   1:  PR[91,3] = PR[90,3] + 83.496;
   1:L PR[91] R[100]mm/sec CNT100;
   1:  PR[91,1] = PR[90,1] + -62.858;
   1:  PR[91,2] = PR[90,2] + -8.805;
   1:  PR[91,3] = PR[90,3] + 83.508;
   1:L PR[91] R[100]mm/sec CNT100;
   1:  PR[91,1] = PR[90,1] + -62.357;
   1:  PR[91,2] = PR[90,2] + -9.939;
   1:  PR[91,3] = PR[90,3] + 83.523;
   1:L PR[91] R[100]mm/sec CNT100;
   1:  PR[91,1] = PR[90,1] + -59.299;
   1:  PR[91,2] = PR[90,2] + -14.135;
   1:  PR[91,3] = PR[90,3] + 83.529;
   1:L PR[91] R[100]mm/sec CNT100;
   1:  PR[91,1] = PR[90,1] + -58.899;
   1:  PR[91,2] = PR[90,2] + -14.496;
   1:  PR[91,3] = PR[90,3] + 83.550;
   1:L PR[91] R[100]mm/sec CNT100;
   1:  PR[91,1] = PR[90,1] + -55.480;
   1:  PR[91,2] = PR[90,2] + -17.247;
   1:  PR[91,3] = PR[90,3] + 83.552;
   1:L PR[91] R[100]mm/sec CNT100;
   1:  PR[91,1] = PR[90,1] + -54.310;
   1:  PR[91,2] = PR[90,2] + -18.147;
   1:  PR[91,3] = PR[90,3] + 83.570;
   1:L PR[91] R[100]mm/sec CNT100;
   1:  PR[91,1] = PR[90,1] + -51.181;
   1:  PR[91,2] = PR[90,2] + -19.877;
   1:  PR[91,3] = PR[90,3] + 83.576;
   1:L PR[91] R[100]mm/sec CNT100;
   1:  PR[91,1] = PR[90,1] + -47.305;
   1:  PR[91,2] = PR[90,2] + -21.893;
   1:  PR[91,3] = PR[90,3] + 83.591;
   1:L PR[91] R[100]mm/sec CNT100;
   1:  PR[91,1] = PR[90,1] + -46.433;
   1:  PR[91,2] = PR[90,2] + -22.219;
   1:  PR[91,3] = PR[90,3] + 83.609;
   1:L PR[91] R[100]mm/sec CNT100;
   1:  PR[91,1] = PR[90,1] + -44.851;
   1:  PR[91,2] = PR[90,2] + -22.759;
   1:  PR[91,3] = PR[90,3] + 83.613;
   1:L PR[91] R[100]mm/sec CNT100;
   1:  PR[91,1] = PR[90,1] + -40.571;
   1:  PR[91,2] = PR[90,2] + -24.060;
   1:  PR[91,3] = PR[90,3] + 83.620;
   1:L PR[91] R[100]mm/sec CNT100;
   1:  PR[91,1] = PR[90,1] + -38.296;
   1:  PR[91,2] = PR[90,2] + -24.719;
   1:  PR[91,3] = PR[90,3] + 83.638;
   1:L PR[91] R[100]mm/sec CNT100;
   1:  PR[91,1] = PR[90,1] + -32.592;
   1:  PR[91,2] = PR[90,2] + -25.826;
   1:  PR[91,3] = PR[90,3] + 83.648;
   1:L PR[91] R[100]mm/sec CNT100;
   1:  PR[91,1] = PR[90,1] + -30.326;
   1:  PR[91,2] = PR[90,2] + -26.230;
   1:  PR[91,3] = PR[90,3] + 83.672;
   1:L PR[91] R[100]mm/sec CNT100;
   1:  PR[91,1] = PR[90,1] + -20.814;
   1:  PR[91,2] = PR[90,2] + -27.225;
   1:  PR[91,3] = PR[90,3] + 83.681;
   1:L PR[91] R[100]mm/sec CNT100;
   1:  PR[91,1] = PR[90,1] + -17.150;
   1:  PR[91,2] = PR[90,2] + -27.366;
   1:  PR[91,3] = PR[90,3] + 83.721;
   1:L PR[91] R[100]mm/sec CNT100;
   1:  PR[91,1] = PR[90,1] + -10.849;
   1:  PR[91,2] = PR[90,2] + -27.576;
   1:  PR[91,3] = PR[90,3] + 83.736;
   1:L PR[91] R[100]mm/sec CNT100;
   1:  PR[91,1] = PR[90,1] + -4.026;
   1:  PR[91,2] = PR[90,2] + -27.361;
   1:  PR[91,3] = PR[90,3] + 83.762;
   1:L PR[91] R[100]mm/sec CNT100;
   1:  PR[91,1] = PR[90,1] + -0.594;
   1:  PR[91,2] = PR[90,2] + -27.232;
   1:  PR[91,3] = PR[90,3] + 83.790;
   1:L PR[91] R[100]mm/sec CNT100;
   1:  PR[91,1] = PR[90,1] + 0.853;
   1:  PR[91,2] = PR[90,2] + -27.123;
   1:  PR[91,3] = PR[90,3] + 83.804;
   1:L PR[91] R[100]mm/sec CNT100;
   1:  PR[91,1] = PR[90,1] + 2.653;
   1:  PR[91,2] = PR[90,2] + -27.252;
   1:  PR[91,3] = PR[90,3] + 83.810;
   1:L PR[91] R[100]mm/sec CNT100;
   1:  PR[91,1] = PR[90,1] + 5.506;
   1:  PR[91,2] = PR[90,2] + -27.258;
   1:  PR[91,3] = PR[90,3] + 83.818;
   1:L PR[91] R[100]mm/sec CNT100;
   1:  PR[91,1] = PR[90,1] + 7.419;
   1:  PR[91,2] = PR[90,2] + -27.285;
   1:  PR[91,3] = PR[90,3] + 83.829;
   1:L PR[91] R[100]mm/sec CNT100;
   1:  PR[91,1] = PR[90,1] + 7.750;
   1:  PR[91,2] = PR[90,2] + -27.279;
   1:  PR[91,3] = PR[90,3] + 83.837;
   1:L PR[91] R[100]mm/sec CNT100;
   1:  PR[91,1] = PR[90,1] + 8.440;
   1:  PR[91,2] = PR[90,2] + -27.232;
   1:  PR[91,3] = PR[90,3] + 83.839;
   1:L PR[91] R[100]mm/sec CNT100;
   1:  PR[91,1] = PR[90,1] + 11.886;
   1:  PR[91,2] = PR[90,2] + -26.903;
   1:  PR[91,3] = PR[90,3] + 83.841;
   1:L PR[91] R[100]mm/sec CNT100;
   1:  PR[91,1] = PR[90,1] + 12.853;
   1:  PR[91,2] = PR[90,2] + -27.102;
   1:  PR[91,3] = PR[90,3] + 83.856;
   1:L PR[91] R[100]mm/sec CNT100;
   1:  PR[91,1] = PR[90,1] + 15.186;
   1:  PR[91,2] = PR[90,2] + -27.492;
   1:  PR[91,3] = PR[90,3] + 83.860;
   1:L PR[91] R[100]mm/sec CNT100;
   1:  PR[91,1] = PR[90,1] + 17.292;
   1:  PR[91,2] = PR[90,2] + -27.750;
   1:  PR[91,3] = PR[90,3] + 83.870;
   1:L PR[91] R[100]mm/sec CNT100;
   1:  PR[91,1] = PR[90,1] + 20.645;
   1:  PR[91,2] = PR[90,2] + -27.636;
   1:  PR[91,3] = PR[90,3] + 83.878;
   1:L PR[91] R[100]mm/sec CNT100;
   1:  PR[91,1] = PR[90,1] + 22.928;
   1:  PR[91,2] = PR[90,2] + -27.593;
   1:  PR[91,3] = PR[90,3] + 83.892;
   1:L PR[91] R[100]mm/sec CNT100;
   1:  PR[91,1] = PR[90,1] + 26.835;
   1:  PR[91,2] = PR[90,2] + -28.529;
   1:  PR[91,3] = PR[90,3] + 83.901;
   1:L PR[91] R[100]mm/sec CNT100;
   1:  PR[91,1] = PR[90,1] + 28.431;
   1:  PR[91,2] = PR[90,2] + -28.891;
   1:  PR[91,3] = PR[90,3] + 83.918;
   1:L PR[91] R[100]mm/sec CNT100;
   1:  PR[91,1] = PR[90,1] + 33.590;
   1:  PR[91,2] = PR[90,2] + -29.193;
   1:  PR[91,3] = PR[90,3] + 83.925;
   1:L PR[91] R[100]mm/sec CNT100;
   1:  PR[91,1] = PR[90,1] + 38.798;
   1:  PR[91,2] = PR[90,2] + -28.611;
   1:  PR[91,3] = PR[90,3] + 83.946;
   1:L PR[91] R[100]mm/sec CNT100;
   1:  PR[91,1] = PR[90,1] + 41.367;
   1:  PR[91,2] = PR[90,2] + -27.900;
   1:  PR[91,3] = PR[90,3] + 83.968;
   1:L PR[91] R[100]mm/sec CNT100;
   1:  PR[91,1] = PR[90,1] + 43.735;
   1:  PR[91,2] = PR[90,2] + -27.217;
   1:  PR[91,3] = PR[90,3] + 83.979;
   1:L PR[91] R[100]mm/sec CNT100;
   1:  PR[91,1] = PR[90,1] + 47.721;
   1:  PR[91,2] = PR[90,2] + -25.319;
   1:  PR[91,3] = PR[90,3] + 83.989;
   1:L PR[91] R[100]mm/sec CNT100;
   1:  PR[91,1] = PR[90,1] + 48.381;
   1:  PR[91,2] = PR[90,2] + -25.044;
   1:  PR[91,3] = PR[90,3] + 84.007;
   1:L PR[91] R[100]mm/sec CNT100;
   1:  PR[91,1] = PR[90,1] + 48.578;
   1:  PR[91,2] = PR[90,2] + -24.941;
   1:  PR[91,3] = PR[90,3] + 84.010;
   1:L PR[91] R[100]mm/sec CNT100;
   1:  PR[91,1] = PR[90,1] + 51.923;
   1:  PR[91,2] = PR[90,2] + -22.835;
   1:  PR[91,3] = PR[90,3] + 84.011;
   1:L PR[91] R[100]mm/sec CNT100;
   1:  PR[91,1] = PR[90,1] + 53.939;
   1:  PR[91,2] = PR[90,2] + -21.330;
   1:  PR[91,3] = PR[90,3] + 84.027;
   1:L PR[91] R[100]mm/sec CNT100;
   1:  PR[91,1] = PR[90,1] + 54.792;
   1:  PR[91,2] = PR[90,2] + -20.561;
   1:  PR[91,3] = PR[90,3] + 84.037;
   1:L PR[91] R[100]mm/sec CNT100;
   1:  PR[91,1] = PR[90,1] + 56.133;
   1:  PR[91,2] = PR[90,2] + -19.163;
   1:  PR[91,3] = PR[90,3] + 84.042;
   1:L PR[91] R[100]mm/sec CNT100;
   1:  PR[91,1] = PR[90,1] + 57.720;
   1:  PR[91,2] = PR[90,2] + -17.820;
   1:  PR[91,3] = PR[90,3] + 84.050;
   1:L PR[91] R[100]mm/sec CNT100;
   1:  PR[91,1] = PR[90,1] + 58.592;
   1:  PR[91,2] = PR[90,2] + -16.934;
   1:  PR[91,3] = PR[90,3] + 84.059;
   1:L PR[91] R[100]mm/sec CNT100;
   1:  PR[91,1] = PR[90,1] + 60.063;
   1:  PR[91,2] = PR[90,2] + -15.177;
   1:  PR[91,3] = PR[90,3] + 84.064;
   1:L PR[91] R[100]mm/sec CNT100;
   1:  PR[91,1] = PR[90,1] + 61.896;
   1:  PR[91,2] = PR[90,2] + -12.606;
   1:  PR[91,3] = PR[90,3] + 84.073;
   1:L PR[91] R[100]mm/sec CNT100;
   1:  PR[91,1] = PR[90,1] + 62.073;
   1:  PR[91,2] = PR[90,2] + -12.393;
   1:  PR[91,3] = PR[90,3] + 84.086;
   1:L PR[91] R[100]mm/sec CNT100;
   1:  PR[91,1] = PR[90,1] + 62.111;
   1:  PR[91,2] = PR[90,2] + -12.327;
   1:  PR[91,3] = PR[90,3] + 84.087;
   1:L PR[91] R[100]mm/sec CNT100;
   1:  PR[91,1] = PR[90,1] + 64.147;
   1:  PR[91,2] = PR[90,2] + -8.707;
   1:  PR[91,3] = PR[90,3] + 84.088;
   1:L PR[91] R[100]mm/sec CNT100;
   1:  PR[91,1] = PR[90,1] + 64.790;
   1:  PR[91,2] = PR[90,2] + -6.800;
   1:  PR[91,3] = PR[90,3] + 84.105;
   1:L PR[91] R[100]mm/sec CNT100;
   1:  PR[91,1] = PR[90,1] + 65.448;
   1:  PR[91,2] = PR[90,2] + -4.780;
   1:  PR[91,3] = PR[90,3] + 84.113;
   1:L PR[91] R[100]mm/sec CNT100;
   1:  PR[91,1] = PR[90,1] + 65.893;
   1:  PR[91,2] = PR[90,2] + -0.729;
   1:  PR[91,3] = PR[90,3] + 84.122;
   1:L PR[91] R[100]mm/sec CNT100;
   1:  PR[91,1] = PR[90,1] + 65.448;
   1:  PR[91,2] = PR[90,2] + 3.322;
   1:  PR[91,3] = PR[90,3] + 84.139;
   1:L PR[91] R[100]mm/sec CNT100;
   1:  PR[91,1] = PR[90,1] + 64.790;
   1:  PR[91,2] = PR[90,2] + 5.341;
   1:  PR[91,3] = PR[90,3] + 84.156;
   1:L PR[91] R[100]mm/sec CNT100;
   1:  PR[91,1] = PR[90,1] + 64.147;
   1:  PR[91,2] = PR[90,2] + 7.247;
   1:  PR[91,3] = PR[90,3] + 84.164;
   1:L PR[91] R[100]mm/sec CNT100;
   1:  PR[91,1] = PR[90,1] + 62.065;
   1:  PR[91,2] = PR[90,2] + 10.944;
   1:  PR[91,3] = PR[90,3] + 84.173;
   1:L PR[91] R[100]mm/sec CNT100;
   1:  PR[91,1] = PR[90,1] + 61.896;
   1:  PR[91,2] = PR[90,2] + 11.147;
   1:  PR[91,3] = PR[90,3] + 84.190;
   1:L PR[91] R[100]mm/sec CNT100;
   1:  PR[91,1] = PR[90,1] + 60.063;
   1:  PR[91,2] = PR[90,2] + 13.718;
   1:  PR[91,3] = PR[90,3] + 84.191;
   1:L PR[91] R[100]mm/sec CNT100;
   1:  PR[91,1] = PR[90,1] + 58.592;
   1:  PR[91,2] = PR[90,2] + 15.476;
   1:  PR[91,3] = PR[90,3] + 84.204;
   1:L PR[91] R[100]mm/sec CNT100;
   1:  PR[91,1] = PR[90,1] + 57.720;
   1:  PR[91,2] = PR[90,2] + 16.362;
   1:  PR[91,3] = PR[90,3] + 84.214;
   1:L PR[91] R[100]mm/sec CNT100;
   1:  PR[91,1] = PR[90,1] + 56.133;
   1:  PR[91,2] = PR[90,2] + 17.704;
   1:  PR[91,3] = PR[90,3] + 84.219;
   1:L PR[91] R[100]mm/sec CNT100;
   1:  PR[91,1] = PR[90,1] + 54.792;
   1:  PR[91,2] = PR[90,2] + 19.102;
   1:  PR[91,3] = PR[90,3] + 84.227;
   1:L PR[91] R[100]mm/sec CNT100;
   1:  PR[91,1] = PR[90,1] + 53.939;
   1:  PR[91,2] = PR[90,2] + 19.872;
   1:  PR[91,3] = PR[90,3] + 84.235;
   1:L PR[91] R[100]mm/sec CNT100;
   1:  PR[91,1] = PR[90,1] + 51.923;
   1:  PR[91,2] = PR[90,2] + 21.376;
   1:  PR[91,3] = PR[90,3] + 84.240;
   1:L PR[91] R[100]mm/sec CNT100;
   1:  PR[91,1] = PR[90,1] + 48.578;
   1:  PR[91,2] = PR[90,2] + 23.482;
   1:  PR[91,3] = PR[90,3] + 84.250;
   1:L PR[91] R[100]mm/sec CNT100;
   1:  PR[91,1] = PR[90,1] + 48.381;
   1:  PR[91,2] = PR[90,2] + 23.585;
   1:  PR[91,3] = PR[90,3] + 84.267;
   1:L PR[91] R[100]mm/sec CNT100;
   1:  PR[91,1] = PR[90,1] + 47.721;
   1:  PR[91,2] = PR[90,2] + 23.860;
   1:  PR[91,3] = PR[90,3] + 84.268;
   1:L PR[91] R[100]mm/sec CNT100;
   1:  PR[91,1] = PR[90,1] + 43.735;
   1:  PR[91,2] = PR[90,2] + 25.759;
   1:  PR[91,3] = PR[90,3] + 84.270;
   1:L PR[91] R[100]mm/sec CNT100;
   1:  PR[91,1] = PR[90,1] + 41.367;
   1:  PR[91,2] = PR[90,2] + 26.441;
   1:  PR[91,3] = PR[90,3] + 84.289;
   1:L PR[91] R[100]mm/sec CNT100;
   1:  PR[91,1] = PR[90,1] + 38.798;
   1:  PR[91,2] = PR[90,2] + 27.152;
   1:  PR[91,3] = PR[90,3] + 84.299;
   1:L PR[91] R[100]mm/sec CNT100;
   1:  PR[91,1] = PR[90,1] + 33.590;
   1:  PR[91,2] = PR[90,2] + 27.734;
   1:  PR[91,3] = PR[90,3] + 84.310;
   1:L PR[91] R[100]mm/sec CNT100;
   1:  PR[91,1] = PR[90,1] + 28.431;
   1:  PR[91,2] = PR[90,2] + 27.432;
   1:  PR[91,3] = PR[90,3] + 84.331;
   1:L PR[91] R[100]mm/sec CNT100;
   1:  PR[91,1] = PR[90,1] + 26.835;
   1:  PR[91,2] = PR[90,2] + 27.070;
   1:  PR[91,3] = PR[90,3] + 84.353;
   1:L PR[91] R[100]mm/sec CNT100;
   1:  PR[91,1] = PR[90,1] + 22.911;
   1:  PR[91,2] = PR[90,2] + 26.131;
   1:  PR[91,3] = PR[90,3] + 84.359;
   1:L PR[91] R[100]mm/sec CNT100;
   1:  PR[91,1] = PR[90,1] + 19.492;
   1:  PR[91,2] = PR[90,2] + 26.252;
   1:  PR[91,3] = PR[90,3] + 84.376;
   1:L PR[91] R[100]mm/sec CNT100;
   1:  PR[91,1] = PR[90,1] + 17.308;
   1:  PR[91,2] = PR[90,2] + 26.293;
   1:  PR[91,3] = PR[90,3] + 84.390;
   1:L PR[91] R[100]mm/sec CNT100;
   1:  PR[91,1] = PR[90,1] + 15.188;
   1:  PR[91,2] = PR[90,2] + 26.034;
   1:  PR[91,3] = PR[90,3] + 84.399;
   1:L PR[91] R[100]mm/sec CNT100;
   1:  PR[91,1] = PR[90,1] + 12.855;
   1:  PR[91,2] = PR[90,2] + 25.644;
   1:  PR[91,3] = PR[90,3] + 84.408;
   1:L PR[91] R[100]mm/sec CNT100;
   1:  PR[91,1] = PR[90,1] + 11.886;
   1:  PR[91,2] = PR[90,2] + 25.445;
   1:  PR[91,3] = PR[90,3] + 84.418;
   1:L PR[91] R[100]mm/sec CNT100;
   1:  PR[91,1] = PR[90,1] + 8.440;
   1:  PR[91,2] = PR[90,2] + 25.773;
   1:  PR[91,3] = PR[90,3] + 84.422;
   1:L PR[91] R[100]mm/sec CNT100;
   1:  PR[91,1] = PR[90,1] + 7.775;
   1:  PR[91,2] = PR[90,2] + 25.818;
   1:  PR[91,3] = PR[90,3] + 84.436;
   1:L PR[91] R[100]mm/sec CNT100;
   1:  PR[91,1] = PR[90,1] + 2.699;
   1:  PR[91,2] = PR[90,2] + 25.794;
   1:  PR[91,3] = PR[90,3] + 84.439;
   1:L PR[91] R[100]mm/sec CNT100;
   1:  PR[91,1] = PR[90,1] + 1.042;
   1:  PR[91,2] = PR[90,2] + 25.626;
   1:  PR[91,3] = PR[90,3] + 84.460;
   1:L PR[91] R[100]mm/sec CNT100;
   1:  PR[91,1] = PR[90,1] + 0.458;
   1:  PR[91,2] = PR[90,2] + 25.698;
   1:  PR[91,3] = PR[90,3] + 84.467;
   1:L PR[91] R[100]mm/sec CNT100;
   1:  PR[91,1] = PR[90,1] + -0.211;
   1:  PR[91,2] = PR[90,2] + 25.747;
   1:  PR[91,3] = PR[90,3] + 84.469;
   1:L PR[91] R[100]mm/sec CNT100;
   1:  PR[91,1] = PR[90,1] + -4.029;
   1:  PR[91,2] = PR[90,2] + 25.902;
   1:  PR[91,3] = PR[90,3] + 84.472;
   1:L PR[91] R[100]mm/sec CNT100;
   1:  PR[91,1] = PR[90,1] + -10.849;
   1:  PR[91,2] = PR[90,2] + 26.117;
   1:  PR[91,3] = PR[90,3] + 84.487;
   1:L PR[91] R[100]mm/sec CNT100;
   1:  PR[91,1] = PR[90,1] + -17.150;
   1:  PR[91,2] = PR[90,2] + 25.907;
   1:  PR[91,3] = PR[90,3] + 84.516;
   1:L PR[91] R[100]mm/sec CNT100;
   1:  PR[91,1] = PR[90,1] + -20.814;
   1:  PR[91,2] = PR[90,2] + 25.766;
   1:  PR[91,3] = PR[90,3] + 84.542;
   1:L PR[91] R[100]mm/sec CNT100;
   1:  PR[91,1] = PR[90,1] + -30.326;
   1:  PR[91,2] = PR[90,2] + 24.771;
   1:  PR[91,3] = PR[90,3] + 84.557;
   1:L PR[91] R[100]mm/sec CNT100;
   1:  PR[91,1] = PR[90,1] + -32.592;
   1:  PR[91,2] = PR[90,2] + 24.367;
   1:  PR[91,3] = PR[90,3] + 84.596;
   1:L PR[91] R[100]mm/sec CNT100;
   1:  PR[91,1] = PR[90,1] + -38.503;
   1:  PR[91,2] = PR[90,2] + 23.224;
   1:  PR[91,3] = PR[90,3] + 84.606;
   1:L PR[91] R[100]mm/sec CNT100;
   1:  PR[91,1] = PR[90,1] + -43.527;
   1:  PR[91,2] = PR[90,2] + 21.723;
   1:  PR[91,3] = PR[90,3] + 84.630;
   1:L PR[91] R[100]mm/sec CNT100;
   1:  PR[91,1] = PR[90,1] + -46.770;
   1:  PR[91,2] = PR[90,2] + 20.639;
   1:  PR[91,3] = PR[90,3] + 84.652;
   1:L PR[91] R[100]mm/sec CNT100;
   1:  PR[91,1] = PR[90,1] + -50.439;
   1:  PR[91,2] = PR[90,2] + 18.870;
   1:  PR[91,3] = PR[90,3] + 84.666;
   1:L PR[91] R[100]mm/sec CNT100;
   1:  PR[91,1] = PR[90,1] + -53.072;
   1:  PR[91,2] = PR[90,2] + 17.528;
   1:  PR[91,3] = PR[90,3] + 84.683;
   1:L PR[91] R[100]mm/sec CNT100;
   1:  PR[91] = PR[90];
   1:  PR[91,1] = PR[90,1] + -56.871;
   1:  PR[91,2] = PR[90,2] + 13.843;
   1:  PR[91,3] = PR[90,3] + 85.995;
   1:L PR[91] R[100]mm/sec CNT100;
   1:  PR[91,1] = PR[90,1] + -57.057;
   1:  PR[91,2] = PR[90,2] + 13.694;
   1:  PR[91,3] = PR[90,3] + 84.721;
   1:L PR[91] R[100]mm/sec CNT100;
   1:  PR[91,1] = PR[90,1] + -60.068;
   1:  PR[91,2] = PR[90,2] + 10.000;
   1:  PR[91,3] = PR[90,3] + 84.722;
   1:L PR[91] R[100]mm/sec CNT100;
   1:  PR[91,1] = PR[90,1] + -60.841;
   1:  PR[91,2] = PR[90,2] + 9.015;
   1:  PR[91,3] = PR[90,3] + 84.742;
   1:L PR[91] R[100]mm/sec CNT100;
   1:  PR[91,1] = PR[90,1] + -62.232;
   1:  PR[91,2] = PR[90,2] + 5.989;
   1:  PR[91,3] = PR[90,3] + 84.747;
   1:L PR[91] R[100]mm/sec CNT100;
   1:  PR[91,1] = PR[90,1] + -63.043;
   1:  PR[91,2] = PR[90,2] + 4.170;
   1:  PR[91,3] = PR[90,3] + 84.761;
   1:L PR[91] R[100]mm/sec CNT100;
   1:  PR[91,1] = PR[90,1] + -63.397;
   1:  PR[91,2] = PR[90,2] + 1.755;
   1:  PR[91,3] = PR[90,3] + 84.770;
   1:L PR[91] R[100]mm/sec CNT100;
   1:  PR[91,1] = PR[90,1] + -63.845;
   1:  PR[91,2] = PR[90,2] + -0.138;
   1:  PR[91,3] = PR[90,3] + 84.780;
   1:L PR[91] R[100]mm/sec CNT100;
   1:  PR[91,1] = PR[90,1] + -63.928;
   1:  PR[91,2] = PR[90,2] + -0.626;
   1:  PR[91,3] = PR[90,3] + 84.788;
   1:L PR[91] R[100]mm/sec CNT100;
   1:  PR[91,1] = PR[90,1] + -63.631;
   1:  PR[91,2] = PR[90,2] + -1.695;
   1:  PR[91,3] = PR[90,3] + 84.790;
   1:L PR[91] R[100]mm/sec CNT100;
   1:  PR[91,1] = PR[90,1] + -63.134;
   1:  PR[91,2] = PR[90,2] + -5.424;
   1:  PR[91,3] = PR[90,3] + 84.795;
   1:L PR[91] R[100]mm/sec CNT100;
   1:  PR[91,1] = PR[90,1] + -61.433;
   1:  PR[91,2] = PR[90,2] + -9.549;
   1:  PR[91,3] = PR[90,3] + 84.810;
   1:L PR[91] R[100]mm/sec CNT100;
   1:  PR[91,1] = PR[90,1] + -61.268;
   1:  PR[91,2] = PR[90,2] + -9.923;
   1:  PR[91,3] = PR[90,3] + 84.829;
   1:L PR[91] R[100]mm/sec CNT100;
   1:  PR[91,1] = PR[90,1] + -59.724;
   1:  PR[91,2] = PR[90,2] + -12.049;
   1:  PR[91,3] = PR[90,3] + 84.831;
   1:L PR[91] R[100]mm/sec CNT100;
   1:  PR[91,1] = PR[90,1] + -57.969;
   1:  PR[91,2] = PR[90,2] + -14.174;
   1:  PR[91,3] = PR[90,3] + 84.842;
   1:L PR[91] R[100]mm/sec CNT100;
   1:  PR[91,1] = PR[90,1] + -54.587;
   1:  PR[91,2] = PR[90,2] + -16.895;
   1:  PR[91,3] = PR[90,3] + 84.853;
   1:L PR[91] R[100]mm/sec CNT100;
   1:  PR[91,1] = PR[90,1] + -52.665;
   1:  PR[91,2] = PR[90,2] + -18.373;
   1:  PR[91,3] = PR[90,3] + 84.871;
   1:L PR[91] R[100]mm/sec CNT100;
   1:  PR[91,1] = PR[90,1] + -50.363;
   1:  PR[91,2] = PR[90,2] + -19.646;
   1:  PR[91,3] = PR[90,3] + 84.881;
   1:L PR[91] R[100]mm/sec CNT100;
   1:  PR[91,1] = PR[90,1] + -45.579;
   1:  PR[91,2] = PR[90,2] + -22.133;
   1:  PR[91,3] = PR[90,3] + 84.892;
   1:L PR[91] R[100]mm/sec CNT100;
   1:  PR[91,1] = PR[90,1] + -39.579;
   1:  PR[91,2] = PR[90,2] + -23.958;
   1:  PR[91,3] = PR[90,3] + 84.915;
   1:L PR[91] R[100]mm/sec CNT100;
   1:  PR[91,1] = PR[90,1] + -36.288;
   1:  PR[91,2] = PR[90,2] + -24.911;
   1:  PR[91,3] = PR[90,3] + 84.941;
   1:L PR[91] R[100]mm/sec CNT100;
   1:  PR[91,1] = PR[90,1] + -33.240;
   1:  PR[91,2] = PR[90,2] + -25.503;
   1:  PR[91,3] = PR[90,3] + 84.955;
   1:L PR[91] R[100]mm/sec CNT100;
   1:  PR[91,1] = PR[90,1] + -27.855;
   1:  PR[91,2] = PR[90,2] + -26.462;
   1:  PR[91,3] = PR[90,3] + 84.968;
   1:L PR[91] R[100]mm/sec CNT100;
   1:  PR[91,1] = PR[90,1] + -18.268;
   1:  PR[91,2] = PR[90,2] + -27.470;
   1:  PR[91,3] = PR[90,3] + 84.991;
   1:L PR[91] R[100]mm/sec CNT100;
   1:  PR[91,1] = PR[90,1] + -13.610;
   1:  PR[91,2] = PR[90,2] + -27.649;
   1:  PR[91,3] = PR[90,3] + 85.031;
   1:L PR[91] R[100]mm/sec CNT100;
   1:  PR[91,1] = PR[90,1] + -8.222;
   1:  PR[91,2] = PR[90,2] + -27.828;
   1:  PR[91,3] = PR[90,3] + 85.051;
   1:L PR[91] R[100]mm/sec CNT100;
   1:  PR[91,1] = PR[90,1] + -0.378;
   1:  PR[91,2] = PR[90,2] + -27.581;
   1:  PR[91,3] = PR[90,3] + 85.073;
   1:L PR[91] R[100]mm/sec CNT100;
   1:  PR[91,1] = PR[90,1] + 2.123;
   1:  PR[91,2] = PR[90,2] + -27.487;
   1:  PR[91,3] = PR[90,3] + 85.106;
   1:L PR[91] R[100]mm/sec CNT100;
   1:  PR[91,1] = PR[90,1] + 2.862;
   1:  PR[91,2] = PR[90,2] + -27.436;
   1:  PR[91,3] = PR[90,3] + 85.116;
   1:L PR[91] R[100]mm/sec CNT100;
   1:  PR[91,1] = PR[90,1] + 3.357;
   1:  PR[91,2] = PR[90,2] + -27.468;
   1:  PR[91,3] = PR[90,3] + 85.119;
   1:L PR[91] R[100]mm/sec CNT100;
   1:  PR[91,1] = PR[90,1] + 7.999;
   1:  PR[91,2] = PR[90,2] + -27.526;
   1:  PR[91,3] = PR[90,3] + 85.122;
   1:L PR[91] R[100]mm/sec CNT100;
   1:  PR[91,1] = PR[90,1] + 8.784;
   1:  PR[91,2] = PR[90,2] + -27.509;
   1:  PR[91,3] = PR[90,3] + 85.141;
   1:L PR[91] R[100]mm/sec CNT100;
   1:  PR[91,1] = PR[90,1] + 10.312;
   1:  PR[91,2] = PR[90,2] + -27.406;
   1:  PR[91,3] = PR[90,3] + 85.144;
   1:L PR[91] R[100]mm/sec CNT100;
   1:  PR[91,1] = PR[90,1] + 12.488;
   1:  PR[91,2] = PR[90,2] + -27.206;
   1:  PR[91,3] = PR[90,3] + 85.151;
   1:L PR[91] R[100]mm/sec CNT100;
   1:  PR[91,1] = PR[90,1] + 14.691;
   1:  PR[91,2] = PR[90,2] + -27.574;
   1:  PR[91,3] = PR[90,3] + 85.160;
   1:L PR[91] R[100]mm/sec CNT100;
   1:  PR[91,1] = PR[90,1] + 17.503;
   1:  PR[91,2] = PR[90,2] + -27.919;
   1:  PR[91,3] = PR[90,3] + 85.169;
   1:L PR[91] R[100]mm/sec CNT100;
   1:  PR[91,1] = PR[90,1] + 19.520;
   1:  PR[91,2] = PR[90,2] + -27.850;
   1:  PR[91,3] = PR[90,3] + 85.181;
   1:L PR[91] R[100]mm/sec CNT100;
   1:  PR[91,1] = PR[90,1] + 22.617;
   1:  PR[91,2] = PR[90,2] + -27.793;
   1:  PR[91,3] = PR[90,3] + 85.189;
   1:L PR[91] R[100]mm/sec CNT100;
   1:  PR[91,1] = PR[90,1] + 25.077;
   1:  PR[91,2] = PR[90,2] + -28.382;
   1:  PR[91,3] = PR[90,3] + 85.202;
   1:L PR[91] R[100]mm/sec CNT100;
   1:  PR[91,1] = PR[90,1] + 26.255;
   1:  PR[91,2] = PR[90,2] + -28.638;
   1:  PR[91,3] = PR[90,3] + 85.213;
   1:L PR[91] R[100]mm/sec CNT100;
   1:  PR[91,1] = PR[90,1] + 28.183;
   1:  PR[91,2] = PR[90,2] + -29.086;
   1:  PR[91,3] = PR[90,3] + 85.218;
   1:L PR[91] R[100]mm/sec CNT100;
   1:  PR[91,1] = PR[90,1] + 33.328;
   1:  PR[91,2] = PR[90,2] + -29.386;
   1:  PR[91,3] = PR[90,3] + 85.226;
   1:L PR[91] R[100]mm/sec CNT100;
   1:  PR[91,1] = PR[90,1] + 35.825;
   1:  PR[91,2] = PR[90,2] + -29.084;
   1:  PR[91,3] = PR[90,3] + 85.247;
   1:L PR[91] R[100]mm/sec CNT100;
   1:  PR[91,1] = PR[90,1] + 38.494;
   1:  PR[91,2] = PR[90,2] + -28.783;
   1:  PR[91,3] = PR[90,3] + 85.258;
   1:L PR[91] R[100]mm/sec CNT100;
   1:  PR[91,1] = PR[90,1] + 39.496;
   1:  PR[91,2] = PR[90,2] + -28.506;
   1:  PR[91,3] = PR[90,3] + 85.269;
   1:L PR[91] R[100]mm/sec CNT100;
   1:  PR[91,1] = PR[90,1] + 43.463;
   1:  PR[91,2] = PR[90,2] + -27.362;
   1:  PR[91,3] = PR[90,3] + 85.273;
   1:L PR[91] R[100]mm/sec CNT100;
   1:  PR[91,1] = PR[90,1] + 48.032;
   1:  PR[91,2] = PR[90,2] + -25.178;
   1:  PR[91,3] = PR[90,3] + 85.291;
   1:L PR[91] R[100]mm/sec CNT100;
   1:  PR[91,1] = PR[90,1] + 49.734;
   1:  PR[91,2] = PR[90,2] + -23.962;
   1:  PR[91,3] = PR[90,3] + 85.312;
   1:L PR[91] R[100]mm/sec CNT100;
   1:  PR[91,1] = PR[90,1] + 51.975;
   1:  PR[91,2] = PR[90,2] + -22.551;
   1:  PR[91,3] = PR[90,3] + 85.321;
   1:L PR[91] R[100]mm/sec CNT100;
   1:  PR[91,1] = PR[90,1] + 52.913;
   1:  PR[91,2] = PR[90,2] + -21.851;
   1:  PR[91,3] = PR[90,3] + 85.332;
   1:L PR[91] R[100]mm/sec CNT100;
   1:  PR[91,1] = PR[90,1] + 54.901;
   1:  PR[91,2] = PR[90,2] + -20.057;
   1:  PR[91,3] = PR[90,3] + 85.336;
   1:L PR[91] R[100]mm/sec CNT100;
   1:  PR[91,1] = PR[90,1] + 57.147;
   1:  PR[91,2] = PR[90,2] + -17.716;
   1:  PR[91,3] = PR[90,3] + 85.348;
   1:L PR[91] R[100]mm/sec CNT100;
   1:  PR[91,1] = PR[90,1] + 57.233;
   1:  PR[91,2] = PR[90,2] + -17.604;
   1:  PR[91,3] = PR[90,3] + 85.361;
   1:L PR[91] R[100]mm/sec CNT100;
   1:  PR[91,1] = PR[90,1] + 57.549;
   1:  PR[91,2] = PR[90,2] + -17.139;
   1:  PR[91,3] = PR[90,3] + 85.362;
   1:L PR[91] R[100]mm/sec CNT100;
   1:  PR[91,1] = PR[90,1] + 59.784;
   1:  PR[91,2] = PR[90,2] + -14.469;
   1:  PR[91,3] = PR[90,3] + 85.364;
   1:L PR[91] R[100]mm/sec CNT100;
   1:  PR[91,1] = PR[90,1] + 60.799;
   1:  PR[91,2] = PR[90,2] + -13.045;
   1:  PR[91,3] = PR[90,3] + 85.379;
   1:L PR[91] R[100]mm/sec CNT100;
   1:  PR[91,1] = PR[90,1] + 61.561;
   1:  PR[91,2] = PR[90,2] + -11.686;
   1:  PR[91,3] = PR[90,3] + 85.386;
   1:L PR[91] R[100]mm/sec CNT100;
   1:  PR[91,1] = PR[90,1] + 62.905;
   1:  PR[91,2] = PR[90,2] + -8.916;
   1:  PR[91,3] = PR[90,3] + 85.392;
   1:L PR[91] R[100]mm/sec CNT100;
   1:  PR[91,1] = PR[90,1] + 63.054;
   1:  PR[91,2] = PR[90,2] + -8.651;
   1:  PR[91,3] = PR[90,3] + 85.405;
   1:L PR[91] R[100]mm/sec CNT100;
   1:  PR[91,1] = PR[90,1] + 64.327;
   1:  PR[91,2] = PR[90,2] + -4.746;
   1:  PR[91,3] = PR[90,3] + 85.407;
   1:L PR[91] R[100]mm/sec CNT100;
   1:  PR[91,1] = PR[90,1] + 64.762;
   1:  PR[91,2] = PR[90,2] + -0.729;
   1:  PR[91,3] = PR[90,3] + 85.424;
   1:L PR[91] R[100]mm/sec CNT100;
   1:  PR[91,1] = PR[90,1] + 64.327;
   1:  PR[91,2] = PR[90,2] + 3.287;
   1:  PR[91,3] = PR[90,3] + 85.441;
   1:L PR[91] R[100]mm/sec CNT100;
   1:  PR[91,1] = PR[90,1] + 63.054;
   1:  PR[91,2] = PR[90,2] + 7.192;
   1:  PR[91,3] = PR[90,3] + 85.457;
   1:L PR[91] R[100]mm/sec CNT100;
   1:  PR[91,1] = PR[90,1] + 62.905;
   1:  PR[91,2] = PR[90,2] + 7.457;
   1:  PR[91,3] = PR[90,3] + 85.474;
   1:L PR[91] R[100]mm/sec CNT100;
   1:  PR[91,1] = PR[90,1] + 61.561;
   1:  PR[91,2] = PR[90,2] + 10.227;
   1:  PR[91,3] = PR[90,3] + 85.476;
   1:L PR[91] R[100]mm/sec CNT100;
   1:  PR[91,1] = PR[90,1] + 60.799;
   1:  PR[91,2] = PR[90,2] + 11.587;
   1:  PR[91,3] = PR[90,3] + 85.489;
   1:L PR[91] R[100]mm/sec CNT100;
   1:  PR[91,1] = PR[90,1] + 59.784;
   1:  PR[91,2] = PR[90,2] + 13.010;
   1:  PR[91,3] = PR[90,3] + 85.495;
   1:L PR[91] R[100]mm/sec CNT100;
   1:  PR[91,1] = PR[90,1] + 57.549;
   1:  PR[91,2] = PR[90,2] + 15.680;
   1:  PR[91,3] = PR[90,3] + 85.502;
   1:L PR[91] R[100]mm/sec CNT100;
   1:  PR[91,1] = PR[90,1] + 57.233;
   1:  PR[91,2] = PR[90,2] + 16.145;
   1:  PR[91,3] = PR[90,3] + 85.517;
   1:L PR[91] R[100]mm/sec CNT100;
   1:  PR[91,1] = PR[90,1] + 57.147;
   1:  PR[91,2] = PR[90,2] + 16.257;
   1:  PR[91,3] = PR[90,3] + 85.519;
   1:L PR[91] R[100]mm/sec CNT100;
   1:  PR[91,1] = PR[90,1] + 54.901;
   1:  PR[91,2] = PR[90,2] + 18.599;
   1:  PR[91,3] = PR[90,3] + 85.520;
   1:L PR[91] R[100]mm/sec CNT100;
   1:  PR[91,1] = PR[90,1] + 52.913;
   1:  PR[91,2] = PR[90,2] + 20.392;
   1:  PR[91,3] = PR[90,3] + 85.533;
   1:L PR[91] R[100]mm/sec CNT100;
   1:  PR[91,1] = PR[90,1] + 51.975;
   1:  PR[91,2] = PR[90,2] + 21.092;
   1:  PR[91,3] = PR[90,3] + 85.545;
   1:L PR[91] R[100]mm/sec CNT100;
   1:  PR[91,1] = PR[90,1] + 49.734;
   1:  PR[91,2] = PR[90,2] + 22.503;
   1:  PR[91,3] = PR[90,3] + 85.549;
   1:L PR[91] R[100]mm/sec CNT100;
   1:  PR[91,1] = PR[90,1] + 48.032;
   1:  PR[91,2] = PR[90,2] + 23.719;
   1:  PR[91,3] = PR[90,3] + 85.560;
   1:L PR[91] R[100]mm/sec CNT100;
   1:  PR[91,1] = PR[90,1] + 43.463;
   1:  PR[91,2] = PR[90,2] + 25.903;
   1:  PR[91,3] = PR[90,3] + 85.569;
   1:L PR[91] R[100]mm/sec CNT100;
   1:  PR[91,1] = PR[90,1] + 39.496;
   1:  PR[91,2] = PR[90,2] + 27.047;
   1:  PR[91,3] = PR[90,3] + 85.590;
   1:L PR[91] R[100]mm/sec CNT100;
   1:  PR[91,1] = PR[90,1] + 38.494;
   1:  PR[91,2] = PR[90,2] + 27.324;
   1:  PR[91,3] = PR[90,3] + 85.608;
   1:L PR[91] R[100]mm/sec CNT100;
   1:  PR[91,1] = PR[90,1] + 35.825;
   1:  PR[91,2] = PR[90,2] + 27.625;
   1:  PR[91,3] = PR[90,3] + 85.612;
   1:L PR[91] R[100]mm/sec CNT100;
   1:  PR[91,1] = PR[90,1] + 33.328;
   1:  PR[91,2] = PR[90,2] + 27.927;
   1:  PR[91,3] = PR[90,3] + 85.623;
   1:L PR[91] R[100]mm/sec CNT100;
   1:  PR[91,1] = PR[90,1] + 28.183;
   1:  PR[91,2] = PR[90,2] + 27.627;
   1:  PR[91,3] = PR[90,3] + 85.634;
   1:L PR[91] R[100]mm/sec CNT100;
   1:  PR[91,1] = PR[90,1] + 26.255;
   1:  PR[91,2] = PR[90,2] + 27.179;
   1:  PR[91,3] = PR[90,3] + 85.655;
   1:L PR[91] R[100]mm/sec CNT100;
   1:  PR[91,1] = PR[90,1] + 25.077;
   1:  PR[91,2] = PR[90,2] + 26.923;
   1:  PR[91,3] = PR[90,3] + 85.663;
   1:L PR[91] R[100]mm/sec CNT100;
   1:  PR[91,1] = PR[90,1] + 22.600;
   1:  PR[91,2] = PR[90,2] + 26.330;
   1:  PR[91,3] = PR[90,3] + 85.668;
   1:L PR[91] R[100]mm/sec CNT100;
   1:  PR[91,1] = PR[90,1] + 20.421;
   1:  PR[91,2] = PR[90,2] + 26.408;
   1:  PR[91,3] = PR[90,3] + 85.679;
   1:L PR[91] R[100]mm/sec CNT100;
   1:  PR[91,1] = PR[90,1] + 17.519;
   1:  PR[91,2] = PR[90,2] + 26.462;
   1:  PR[91,3] = PR[90,3] + 85.688;
   1:L PR[91] R[100]mm/sec CNT100;
   1:  PR[91,1] = PR[90,1] + 14.694;
   1:  PR[91,2] = PR[90,2] + 26.116;
   1:  PR[91,3] = PR[90,3] + 85.700;
   1:L PR[91] R[100]mm/sec CNT100;
   1:  PR[91,1] = PR[90,1] + 12.488;
   1:  PR[91,2] = PR[90,2] + 25.747;
   1:  PR[91,3] = PR[90,3] + 85.712;
   1:L PR[91] R[100]mm/sec CNT100;
   1:  PR[91,1] = PR[90,1] + 10.311;
   1:  PR[91,2] = PR[90,2] + 25.948;
   1:  PR[91,3] = PR[90,3] + 85.721;
   1:L PR[91] R[100]mm/sec CNT100;
   1:  PR[91,1] = PR[90,1] + 8.810;
   1:  PR[91,2] = PR[90,2] + 26.049;
   1:  PR[91,3] = PR[90,3] + 85.731;
   1:L PR[91] R[100]mm/sec CNT100;
   1:  PR[91,1] = PR[90,1] + 3.401;
   1:  PR[91,2] = PR[90,2] + 26.009;
   1:  PR[91,3] = PR[90,3] + 85.737;
   1:L PR[91] R[100]mm/sec CNT100;
   1:  PR[91,1] = PR[90,1] + 2.940;
   1:  PR[91,2] = PR[90,2] + 25.963;
   1:  PR[91,3] = PR[90,3] + 85.759;
   1:L PR[91] R[100]mm/sec CNT100;
   1:  PR[91,1] = PR[90,1] + 2.522;
   1:  PR[91,2] = PR[90,2] + 26.001;
   1:  PR[91,3] = PR[90,3] + 85.761;
   1:L PR[91] R[100]mm/sec CNT100;
   1:  PR[91,1] = PR[90,1] + -0.383;
   1:  PR[91,2] = PR[90,2] + 26.122;
   1:  PR[91,3] = PR[90,3] + 85.763;
   1:L PR[91] R[100]mm/sec CNT100;
   1:  PR[91,1] = PR[90,1] + -8.222;
   1:  PR[91,2] = PR[90,2] + 26.369;
   1:  PR[91,3] = PR[90,3] + 85.775;
   1:L PR[91] R[100]mm/sec CNT100;
   1:  PR[91,1] = PR[90,1] + -13.610;
   1:  PR[91,2] = PR[90,2] + 26.190;
   1:  PR[91,3] = PR[90,3] + 85.808;
   1:L PR[91] R[100]mm/sec CNT100;
   1:  PR[91,1] = PR[90,1] + -18.268;
   1:  PR[91,2] = PR[90,2] + 26.011;
   1:  PR[91,3] = PR[90,3] + 85.830;
   1:L PR[91] R[100]mm/sec CNT100;
   1:  PR[91,1] = PR[90,1] + -27.855;
   1:  PR[91,2] = PR[90,2] + 25.003;
   1:  PR[91,3] = PR[90,3] + 85.850;
   1:L PR[91] R[100]mm/sec CNT100;
   1:  PR[91,1] = PR[90,1] + -33.241;
   1:  PR[91,2] = PR[90,2] + 24.044;
   1:  PR[91,3] = PR[90,3] + 85.890;
   1:L PR[91] R[100]mm/sec CNT100;
   1:  PR[91,1] = PR[90,1] + -36.397;
   1:  PR[91,2] = PR[90,2] + 23.433;
   1:  PR[91,3] = PR[90,3] + 85.913;
   1:L PR[91] R[100]mm/sec CNT100;
   1:  PR[91,1] = PR[90,1] + -44.365;
   1:  PR[91,2] = PR[90,2] + 21.053;
   1:  PR[91,3] = PR[90,3] + 85.926;
   1:L PR[91] R[100]mm/sec CNT100;
   1:  PR[91,1] = PR[90,1] + -45.496;
   1:  PR[91,2] = PR[90,2] + 20.675;
   1:  PR[91,3] = PR[90,3] + 85.961;
   1:L PR[91] R[100]mm/sec CNT100;
   1:  PR[91,1] = PR[90,1] + -46.798;
   1:  PR[91,2] = PR[90,2] + 20.047;
   1:  PR[91,3] = PR[90,3] + 85.966;
   1:L PR[91] R[100]mm/sec CNT100;
   1:  PR[91,1] = PR[90,1] + -51.729;
   1:  PR[91,2] = PR[90,2] + 17.534;
   1:  PR[91,3] = PR[90,3] + 85.972;
   1:L PR[91] R[100]mm/sec CNT100;
   1:  PR[91] = PR[90];
   1:  PR[91,1] = PR[90,1] + -54.557;
   1:  PR[91,2] = PR[90,2] + 14.545;
   1:  PR[91,3] = PR[90,3] + 87.295;
   1:L PR[91] R[100]mm/sec CNT100;
   1:  PR[91,1] = PR[90,1] + -55.732;
   1:  PR[91,2] = PR[90,2] + 13.660;
   1:  PR[91,3] = PR[90,3] + 86.017;
   1:L PR[91] R[100]mm/sec CNT100;
   1:  PR[91,1] = PR[90,1] + -57.619;
   1:  PR[91,2] = PR[90,2] + 11.580;
   1:  PR[91,3] = PR[90,3] + 86.023;
   1:L PR[91] R[100]mm/sec CNT100;
   1:  PR[91,1] = PR[90,1] + -59.303;
   1:  PR[91,2] = PR[90,2] + 9.513;
   1:  PR[91,3] = PR[90,3] + 86.035;
   1:L PR[91] R[100]mm/sec CNT100;
   1:  PR[91,1] = PR[90,1] + -59.600;
   1:  PR[91,2] = PR[90,2] + 9.136;
   1:  PR[91,3] = PR[90,3] + 86.046;
   1:L PR[91] R[100]mm/sec CNT100;
   1:  PR[91,1] = PR[90,1] + -61.331;
   1:  PR[91,2] = PR[90,2] + 5.370;
   1:  PR[91,3] = PR[90,3] + 86.048;
   1:L PR[91] R[100]mm/sec CNT100;
   1:  PR[91,1] = PR[90,1] + -61.838;
   1:  PR[91,2] = PR[90,2] + 4.232;
   1:  PR[91,3] = PR[90,3] + 86.066;
   1:L PR[91] R[100]mm/sec CNT100;
   1:  PR[91,1] = PR[90,1] + -62.067;
   1:  PR[91,2] = PR[90,2] + 2.669;
   1:  PR[91,3] = PR[90,3] + 86.071;
   1:L PR[91] R[100]mm/sec CNT100;
   1:  PR[91,1] = PR[90,1] + -62.370;
   1:  PR[91,2] = PR[90,2] + 1.388;
   1:  PR[91,3] = PR[90,3] + 86.077;
   1:L PR[91] R[100]mm/sec CNT100;
   1:  PR[91,1] = PR[90,1] + -62.716;
   1:  PR[91,2] = PR[90,2] + -0.626;
   1:  PR[91,3] = PR[90,3] + 86.083;
   1:L PR[91] R[100]mm/sec CNT100;
   1:  PR[91,1] = PR[90,1] + -62.606;
   1:  PR[91,2] = PR[90,2] + -1.023;
   1:  PR[91,3] = PR[90,3] + 86.092;
   1:L PR[91] R[100]mm/sec CNT100;
   1:  PR[91,1] = PR[90,1] + -62.021;
   1:  PR[91,2] = PR[90,2] + -5.413;
   1:  PR[91,3] = PR[90,3] + 86.093;
   1:L PR[91] R[100]mm/sec CNT100;
   1:  PR[91,1] = PR[90,1] + -60.584;
   1:  PR[91,2] = PR[90,2] + -8.897;
   1:  PR[91,3] = PR[90,3] + 86.112;
   1:L PR[91] R[100]mm/sec CNT100;
   1:  PR[91,1] = PR[90,1] + -60.130;
   1:  PR[91,2] = PR[90,2] + -9.863;
   1:  PR[91,3] = PR[90,3] + 86.128;
   1:L PR[91] R[100]mm/sec CNT100;
   1:  PR[91,1] = PR[90,1] + -57.250;
   1:  PR[91,2] = PR[90,2] + -13.376;
   1:  PR[91,3] = PR[90,3] + 86.132;
   1:L PR[91] R[100]mm/sec CNT100;
   1:  PR[91,1] = PR[90,1] + -56.430;
   1:  PR[91,2] = PR[90,2] + -14.341;
   1:  PR[91,3] = PR[90,3] + 86.152;
   1:L PR[91] R[100]mm/sec CNT100;
   1:  PR[91,1] = PR[90,1] + -53.694;
   1:  PR[91,2] = PR[90,2] + -16.543;
   1:  PR[91,3] = PR[90,3] + 86.157;
   1:L PR[91] R[100]mm/sec CNT100;
   1:  PR[91,1] = PR[90,1] + -51.020;
   1:  PR[91,2] = PR[90,2] + -18.600;
   1:  PR[91,3] = PR[90,3] + 86.172;
   1:L PR[91] R[100]mm/sec CNT100;
   1:  PR[91,1] = PR[90,1] + -49.545;
   1:  PR[91,2] = PR[90,2] + -19.415;
   1:  PR[91,3] = PR[90,3] + 86.186;
   1:L PR[91] R[100]mm/sec CNT100;
   1:  PR[91,1] = PR[90,1] + -46.306;
   1:  PR[91,2] = PR[90,2] + -21.100;
   1:  PR[91,3] = PR[90,3] + 86.193;
   1:L PR[91] R[100]mm/sec CNT100;
   1:  PR[91,1] = PR[90,1] + -44.275;
   1:  PR[91,2] = PR[90,2] + -22.033;
   1:  PR[91,3] = PR[90,3] + 86.209;
   1:L PR[91] R[100]mm/sec CNT100;
   1:  PR[91,1] = PR[90,1] + -43.151;
   1:  PR[91,2] = PR[90,2] + -22.468;
   1:  PR[91,3] = PR[90,3] + 86.218;
   1:L PR[91] R[100]mm/sec CNT100;
   1:  PR[91,1] = PR[90,1] + -38.587;
   1:  PR[91,2] = PR[90,2] + -23.856;
   1:  PR[91,3] = PR[90,3] + 86.223;
   1:L PR[91] R[100]mm/sec CNT100;
   1:  PR[91,1] = PR[90,1] + -34.294;
   1:  PR[91,2] = PR[90,2] + -25.099;
   1:  PR[91,3] = PR[90,3] + 86.243;
   1:L PR[91] R[100]mm/sec CNT100;
   1:  PR[91,1] = PR[90,1] + -25.383;
   1:  PR[91,2] = PR[90,2] + -26.694;
   1:  PR[91,3] = PR[90,3] + 86.262;
   1:L PR[91] R[100]mm/sec CNT100;
   1:  PR[91,1] = PR[90,1] + -15.722;
   1:  PR[91,2] = PR[90,2] + -27.714;
   1:  PR[91,3] = PR[90,3] + 86.300;
   1:L PR[91] R[100]mm/sec CNT100;
   1:  PR[91,1] = PR[90,1] + -10.070;
   1:  PR[91,2] = PR[90,2] + -27.932;
   1:  PR[91,3] = PR[90,3] + 86.341;
   1:L PR[91] R[100]mm/sec CNT100;
   1:  PR[91,1] = PR[90,1] + -5.595;
   1:  PR[91,2] = PR[90,2] + -28.081;
   1:  PR[91,3] = PR[90,3] + 86.365;
   1:L PR[91] R[100]mm/sec CNT100;
   1:  PR[91,1] = PR[90,1] + 3.264;
   1:  PR[91,2] = PR[90,2] + -27.801;
   1:  PR[91,3] = PR[90,3] + 86.384;
   1:L PR[91] R[100]mm/sec CNT100;
   1:  PR[91,1] = PR[90,1] + 5.227;
   1:  PR[91,2] = PR[90,2] + -27.718;
   1:  PR[91,3] = PR[90,3] + 86.422;
   1:L PR[91] R[100]mm/sec CNT100;
   1:  PR[91,1] = PR[90,1] + 8.583;
   1:  PR[91,2] = PR[90,2] + -27.766;
   1:  PR[91,3] = PR[90,3] + 86.430;
   1:L PR[91] R[100]mm/sec CNT100;
   1:  PR[91,1] = PR[90,1] + 9.829;
   1:  PR[91,2] = PR[90,2] + -27.740;
   1:  PR[91,3] = PR[90,3] + 86.444;
   1:L PR[91] R[100]mm/sec CNT100;
   1:  PR[91,1] = PR[90,1] + 11.028;
   1:  PR[91,2] = PR[90,2] + -27.673;
   1:  PR[91,3] = PR[90,3] + 86.449;
   1:L PR[91] R[100]mm/sec CNT100;
   1:  PR[91,1] = PR[90,1] + 13.197;
   1:  PR[91,2] = PR[90,2] + -27.489;
   1:  PR[91,3] = PR[90,3] + 86.454;
   1:L PR[91] R[100]mm/sec CNT100;
   1:  PR[91,1] = PR[90,1] + 14.197;
   1:  PR[91,2] = PR[90,2] + -27.656;
   1:  PR[91,3] = PR[90,3] + 86.464;
   1:L PR[91] R[100]mm/sec CNT100;
   1:  PR[91,1] = PR[90,1] + 17.715;
   1:  PR[91,2] = PR[90,2] + -28.088;
   1:  PR[91,3] = PR[90,3] + 86.468;
   1:L PR[91] R[100]mm/sec CNT100;
   1:  PR[91,1] = PR[90,1] + 18.395;
   1:  PR[91,2] = PR[90,2] + -28.064;
   1:  PR[91,3] = PR[90,3] + 86.483;
   1:L PR[91] R[100]mm/sec CNT100;
   1:  PR[91,1] = PR[90,1] + 22.306;
   1:  PR[91,2] = PR[90,2] + -27.992;
   1:  PR[91,3] = PR[90,3] + 86.486;
   1:L PR[91] R[100]mm/sec CNT100;
   1:  PR[91,1] = PR[90,1] + 23.329;
   1:  PR[91,2] = PR[90,2] + -28.237;
   1:  PR[91,3] = PR[90,3] + 86.502;
   1:L PR[91] R[100]mm/sec CNT100;
   1:  PR[91,1] = PR[90,1] + 25.049;
   1:  PR[91,2] = PR[90,2] + -28.611;
   1:  PR[91,3] = PR[90,3] + 86.507;
   1:L PR[91] R[100]mm/sec CNT100;
   1:  PR[91,1] = PR[90,1] + 27.930;
   1:  PR[91,2] = PR[90,2] + -29.280;
   1:  PR[91,3] = PR[90,3] + 86.514;
   1:L PR[91] R[100]mm/sec CNT100;
   1:  PR[91,1] = PR[90,1] + 33.107;
   1:  PR[91,2] = PR[90,2] + -29.577;
   1:  PR[91,3] = PR[90,3] + 86.527;
   1:L PR[91] R[100]mm/sec CNT100;
   1:  PR[91,1] = PR[90,1] + 38.187;
   1:  PR[91,2] = PR[90,2] + -28.964;
   1:  PR[91,3] = PR[90,3] + 86.548;
   1:L PR[91] R[100]mm/sec CNT100;
   1:  PR[91,1] = PR[90,1] + 38.984;
   1:  PR[91,2] = PR[90,2] + -28.719;
   1:  PR[91,3] = PR[90,3] + 86.570;
   1:L PR[91] R[100]mm/sec CNT100;
   1:  PR[91,1] = PR[90,1] + 43.191;
   1:  PR[91,2] = PR[90,2] + -27.507;
   1:  PR[91,3] = PR[90,3] + 86.574;
   1:L PR[91] R[100]mm/sec CNT100;
   1:  PR[91,1] = PR[90,1] + 47.791;
   1:  PR[91,2] = PR[90,2] + -25.296;
   1:  PR[91,3] = PR[90,3] + 86.592;
   1:L PR[91] R[100]mm/sec CNT100;
   1:  PR[91,1] = PR[90,1] + 51.906;
   1:  PR[91,2] = PR[90,2] + -22.353;
   1:  PR[91,3] = PR[90,3] + 86.614;
   1:L PR[91] R[100]mm/sec CNT100;
   1:  PR[91,1] = PR[90,1] + 55.009;
   1:  PR[91,2] = PR[90,2] + -19.554;
   1:  PR[91,3] = PR[90,3] + 86.635;
   1:L PR[91] R[100]mm/sec CNT100;
   1:  PR[91,1] = PR[90,1] + 56.295;
   1:  PR[91,2] = PR[90,2] + -18.214;
   1:  PR[91,3] = PR[90,3] + 86.653;
   1:L PR[91] R[100]mm/sec CNT100;
   1:  PR[91,1] = PR[90,1] + 57.361;
   1:  PR[91,2] = PR[90,2] + -16.831;
   1:  PR[91,3] = PR[90,3] + 86.660;
   1:L PR[91] R[100]mm/sec CNT100;
   1:  PR[91,1] = PR[90,1] + 59.192;
   1:  PR[91,2] = PR[90,2] + -14.135;
   1:  PR[91,3] = PR[90,3] + 86.668;
   1:L PR[91] R[100]mm/sec CNT100;
   1:  PR[91,1] = PR[90,1] + 59.505;
   1:  PR[91,2] = PR[90,2] + -13.760;
   1:  PR[91,3] = PR[90,3] + 86.682;
   1:L PR[91] R[100]mm/sec CNT100;
   1:  PR[91,1] = PR[90,1] + 59.548;
   1:  PR[91,2] = PR[90,2] + -13.700;
   1:  PR[91,3] = PR[90,3] + 86.684;
   1:L PR[91] R[100]mm/sec CNT100;
   1:  PR[91,1] = PR[90,1] + 61.254;
   1:  PR[91,2] = PR[90,2] + -10.656;
   1:L PR[91] R[100]mm/sec CNT100;
   1:  PR[91,1] = PR[90,1] + 61.997;
   1:  PR[91,2] = PR[90,2] + -9.125;
   1:  PR[91,3] = PR[90,3] + 86.699;
   1:L PR[91] R[100]mm/sec CNT100;
   1:  PR[91,1] = PR[90,1] + 62.495;
   1:  PR[91,2] = PR[90,2] + -7.575;
   1:  PR[91,3] = PR[90,3] + 86.706;
   1:L PR[91] R[100]mm/sec CNT100;
   1:  PR[91,1] = PR[90,1] + 63.268;
   1:  PR[91,2] = PR[90,2] + -4.845;
   1:  PR[91,3] = PR[90,3] + 86.713;
   1:L PR[91] R[100]mm/sec CNT100;
   1:  PR[91,1] = PR[90,1] + 63.661;
   1:  PR[91,2] = PR[90,2] + -0.729;
   1:  PR[91,3] = PR[90,3] + 86.725;
   1:L PR[91] R[100]mm/sec CNT100;
   1:  PR[91,1] = PR[90,1] + 63.268;
   1:  PR[91,2] = PR[90,2] + 3.386;
   1:  PR[91,3] = PR[90,3] + 86.742;
   1:L PR[91] R[100]mm/sec CNT100;
   1:  PR[91,1] = PR[90,1] + 62.495;
   1:  PR[91,2] = PR[90,2] + 6.116;
   1:  PR[91,3] = PR[90,3] + 86.760;
   1:L PR[91] R[100]mm/sec CNT100;
   1:  PR[91,1] = PR[90,1] + 61.997;
   1:  PR[91,2] = PR[90,2] + 7.666;
   1:  PR[91,3] = PR[90,3] + 86.772;
   1:L PR[91] R[100]mm/sec CNT100;
   1:  PR[91,1] = PR[90,1] + 61.254;
   1:  PR[91,2] = PR[90,2] + 9.197;
   1:  PR[91,3] = PR[90,3] + 86.778;
   1:L PR[91] R[100]mm/sec CNT100;
   1:  PR[91,1] = PR[90,1] + 59.548;
   1:  PR[91,2] = PR[90,2] + 12.241;
   1:  PR[91,3] = PR[90,3] + 86.786;
   1:L PR[91] R[100]mm/sec CNT100;
   1:  PR[91,1] = PR[90,1] + 59.505;
   1:  PR[91,2] = PR[90,2] + 12.302;
   1:  PR[91,3] = PR[90,3] + 86.800;
   1:L PR[91] R[100]mm/sec CNT100;
   1:  PR[91,1] = PR[90,1] + 59.192;
   1:  PR[91,2] = PR[90,2] + 12.676;
   1:  PR[91,3] = PR[90,3] + 86.801;
   1:L PR[91] R[100]mm/sec CNT100;
   1:  PR[91,1] = PR[90,1] + 57.361;
   1:  PR[91,2] = PR[90,2] + 15.372;
   1:  PR[91,3] = PR[90,3] + 86.803;
   1:L PR[91] R[100]mm/sec CNT100;
   1:  PR[91,1] = PR[90,1] + 56.295;
   1:  PR[91,2] = PR[90,2] + 16.755;
   1:  PR[91,3] = PR[90,3] + 86.816;
   1:L PR[91] R[100]mm/sec CNT100;
   1:  PR[91,1] = PR[90,1] + 55.009;
   1:  PR[91,2] = PR[90,2] + 18.095;
   1:  PR[91,3] = PR[90,3] + 86.824;
   1:L PR[91] R[100]mm/sec CNT100;
   1:  PR[91,1] = PR[90,1] + 51.901;
   1:  PR[91,2] = PR[90,2] + 20.899;
   1:  PR[91,3] = PR[90,3] + 86.832;
   1:L PR[91] R[100]mm/sec CNT100;
   1:  PR[91,1] = PR[90,1] + 47.791;
   1:  PR[91,2] = PR[90,2] + 23.837;
   1:  PR[91,3] = PR[90,3] + 86.849;
   1:L PR[91] R[100]mm/sec CNT100;
   1:  PR[91,1] = PR[90,1] + 43.191;
   1:  PR[91,2] = PR[90,2] + 26.048;
   1:  PR[91,3] = PR[90,3] + 86.871;
   1:L PR[91] R[100]mm/sec CNT100;
   1:  PR[91,1] = PR[90,1] + 38.984;
   1:  PR[91,2] = PR[90,2] + 27.261;
   1:  PR[91,3] = PR[90,3] + 86.892;
   1:L PR[91] R[100]mm/sec CNT100;
   1:  PR[91,1] = PR[90,1] + 38.187;
   1:  PR[91,2] = PR[90,2] + 27.505;
   1:  PR[91,3] = PR[90,3] + 86.911;
   1:L PR[91] R[100]mm/sec CNT100;
   1:  PR[91,1] = PR[90,1] + 33.107;
   1:  PR[91,2] = PR[90,2] + 28.118;
   1:  PR[91,3] = PR[90,3] + 86.914;
   1:L PR[91] R[100]mm/sec CNT100;
   1:  PR[91,1] = PR[90,1] + 27.930;
   1:  PR[91,2] = PR[90,2] + 27.821;
   1:  PR[91,3] = PR[90,3] + 86.936;
   1:L PR[91] R[100]mm/sec CNT100;
   1:  PR[91,1] = PR[90,1] + 25.049;
   1:  PR[91,2] = PR[90,2] + 27.153;
   1:  PR[91,3] = PR[90,3] + 86.958;
   1:L PR[91] R[100]mm/sec CNT100;
   1:  PR[91,1] = PR[90,1] + 23.328;
   1:  PR[91,2] = PR[90,2] + 26.778;
   1:  PR[91,3] = PR[90,3] + 86.970;
   1:L PR[91] R[100]mm/sec CNT100;
   1:  PR[91,1] = PR[90,1] + 22.303;
   1:  PR[91,2] = PR[90,2] + 26.533;
   1:  PR[91,3] = PR[90,3] + 86.978;
   1:L PR[91] R[100]mm/sec CNT100;
   1:  PR[91,1] = PR[90,1] + 17.727;
   1:  PR[91,2] = PR[90,2] + 26.631;
   1:  PR[91,3] = PR[90,3] + 86.982;
   1:L PR[91] R[100]mm/sec CNT100;
   1:  PR[91,1] = PR[90,1] + 14.200;
   1:  PR[91,2] = PR[90,2] + 26.198;
   1:  PR[91,3] = PR[90,3] + 87.001;
   1:L PR[91] R[100]mm/sec CNT100;
   1:  PR[91,1] = PR[90,1] + 13.197;
   1:  PR[91,2] = PR[90,2] + 26.031;
   1:  PR[91,3] = PR[90,3] + 87.016;
   1:L PR[91] R[100]mm/sec CNT100;
   1:  PR[91,1] = PR[90,1] + 11.029;
   1:  PR[91,2] = PR[90,2] + 26.214;
   1:  PR[91,3] = PR[90,3] + 87.021;
   1:L PR[91] R[100]mm/sec CNT100;
   1:  PR[91,1] = PR[90,1] + 9.854;
   1:  PR[91,2] = PR[90,2] + 26.280;
   1:  PR[91,3] = PR[90,3] + 87.030;
   1:L PR[91] R[100]mm/sec CNT100;
   1:  PR[91,1] = PR[90,1] + 5.422;
   1:  PR[91,2] = PR[90,2] + 26.244;
   1:  PR[91,3] = PR[90,3] + 87.035;
   1:L PR[91] R[100]mm/sec CNT100;
   1:  PR[91,1] = PR[90,1] + 3.261;
   1:  PR[91,2] = PR[90,2] + 26.343;
   1:  PR[91,3] = PR[90,3] + 87.054;
   1:L PR[91] R[100]mm/sec CNT100;
   1:  PR[91,1] = PR[90,1] + -5.595;
   1:  PR[91,2] = PR[90,2] + 26.622;
   1:  PR[91,3] = PR[90,3] + 87.063;
   1:L PR[91] R[100]mm/sec CNT100;
   1:  PR[91,1] = PR[90,1] + -10.070;
   1:  PR[91,2] = PR[90,2] + 26.473;
   1:  PR[91,3] = PR[90,3] + 87.100;
   1:L PR[91] R[100]mm/sec CNT100;
   1:  PR[91,1] = PR[90,1] + -15.722;
   1:  PR[91,2] = PR[90,2] + 26.255;
   1:  PR[91,3] = PR[90,3] + 87.119;
   1:L PR[91] R[100]mm/sec CNT100;
   1:  PR[91,1] = PR[90,1] + -25.383;
   1:  PR[91,2] = PR[90,2] + 25.236;
   1:  PR[91,3] = PR[90,3] + 87.143;
   1:L PR[91] R[100]mm/sec CNT100;
   1:  PR[91,1] = PR[90,1] + -34.305;
   1:  PR[91,2] = PR[90,2] + 23.639;
   1:  PR[91,3] = PR[90,3] + 87.184;
   1:L PR[91] R[100]mm/sec CNT100;
   1:  PR[91,1] = PR[90,1] + -43.755;
   1:  PR[91,2] = PR[90,2] + 20.827;
   1:  PR[91,3] = PR[90,3] + 87.222;
   1:L PR[91] R[100]mm/sec CNT100;
   1:  PR[91,1] = PR[90,1] + -44.200;
   1:  PR[91,2] = PR[90,2] + 20.657;
   1:  PR[91,3] = PR[90,3] + 87.264;
   1:L PR[91] R[100]mm/sec CNT100;
   1:  PR[91,1] = PR[90,1] + -44.933;
   1:  PR[91,2] = PR[90,2] + 20.319;
   1:  PR[91,3] = PR[90,3] + 87.266;
   1:L PR[91] R[100]mm/sec CNT100;
   1:  PR[91,1] = PR[90,1] + -50.386;
   1:  PR[91,2] = PR[90,2] + 17.540;
   1:  PR[91,3] = PR[90,3] + 87.269;
   1:L PR[91] R[100]mm/sec CNT100;
   1:  PR[91] = PR[90];
   1:  PR[91,1] = PR[90,1] + -51.542;
   1:  PR[91,2] = PR[90,2] + 15.752;
   1:  PR[91,3] = PR[90,3] + 88.595;
   1:L PR[91] R[100]mm/sec CNT100;
   1:  PR[91,1] = PR[90,1] + -54.329;
   1:  PR[91,2] = PR[90,2] + 13.650;
   1:  PR[91,3] = PR[90,3] + 87.308;
   1:L PR[91] R[100]mm/sec CNT100;
   1:  PR[91,1] = PR[90,1] + -58.402;
   1:  PR[91,2] = PR[90,2] + 9.161;
   1:  PR[91,3] = PR[90,3] + 87.323;
   1:L PR[91] R[100]mm/sec CNT100;
   1:  PR[91,1] = PR[90,1] + -60.635;
   1:  PR[91,2] = PR[90,2] + 4.283;
   1:  PR[91,3] = PR[90,3] + 87.349;
   1:L PR[91] R[100]mm/sec CNT100;
   1:  PR[91,1] = PR[90,1] + -60.738;
   1:  PR[91,2] = PR[90,2] + 3.582;
   1:  PR[91,3] = PR[90,3] + 87.372;
   1:L PR[91] R[100]mm/sec CNT100;
   1:  PR[91,1] = PR[90,1] + -60.896;
   1:  PR[91,2] = PR[90,2] + 2.913;
   1:  PR[91,3] = PR[90,3] + 87.375;
   1:L PR[91] R[100]mm/sec CNT100;
   1:  PR[91,1] = PR[90,1] + -61.524;
   1:  PR[91,2] = PR[90,2] + -0.747;
   1:  PR[91,3] = PR[90,3] + 87.378;
   1:L PR[91] R[100]mm/sec CNT100;
   1:  PR[91,1] = PR[90,1] + -60.955;
   1:  PR[91,2] = PR[90,2] + -4.707;
   1:  PR[91,3] = PR[90,3] + 87.394;
   1:L PR[91] R[100]mm/sec CNT100;
   1:  PR[91,1] = PR[90,1] + -60.838;
   1:  PR[91,2] = PR[90,2] + -5.325;
   1:  PR[91,3] = PR[90,3] + 87.411;
   1:L PR[91] R[100]mm/sec CNT100;
   1:  PR[91,1] = PR[90,1] + -58.970;
   1:  PR[91,2] = PR[90,2] + -9.317;
   1:  PR[91,3] = PR[90,3] + 87.413;
   1:L PR[91] R[100]mm/sec CNT100;
   1:  PR[91,1] = PR[90,1] + -58.652;
   1:  PR[91,2] = PR[90,2] + -9.976;
   1:  PR[91,3] = PR[90,3] + 87.432;
   1:L PR[91] R[100]mm/sec CNT100;
   1:  PR[91,1] = PR[90,1] + -56.254;
   1:  PR[91,2] = PR[90,2] + -12.901;
   1:  PR[91,3] = PR[90,3] + 87.435;
   1:L PR[91] R[100]mm/sec CNT100;
   1:  PR[91,1] = PR[90,1] + -54.881;
   1:  PR[91,2] = PR[90,2] + -14.517;
   1:  PR[91,3] = PR[90,3] + 87.451;
   1:L PR[91] R[100]mm/sec CNT100;
   1:  PR[91,1] = PR[90,1] + -52.801;
   1:  PR[91,2] = PR[90,2] + -16.191;
   1:  PR[91,3] = PR[90,3] + 87.460;
   1:L PR[91] R[100]mm/sec CNT100;
   1:  PR[91,1] = PR[90,1] + -49.375;
   1:  PR[91,2] = PR[90,2] + -18.826;
   1:  PR[91,3] = PR[90,3] + 87.472;
   1:L PR[91] R[100]mm/sec CNT100;
   1:  PR[91,1] = PR[90,1] + -48.727;
   1:  PR[91,2] = PR[90,2] + -19.184;
   1:  PR[91,3] = PR[90,3] + 87.490;
   1:L PR[91] R[100]mm/sec CNT100;
   1:  PR[91,1] = PR[90,1] + -47.166;
   1:  PR[91,2] = PR[90,2] + -19.996;
   1:  PR[91,3] = PR[90,3] + 87.493;
   1:L PR[91] R[100]mm/sec CNT100;
   1:  PR[91,1] = PR[90,1] + -42.988;
   1:  PR[91,2] = PR[90,2] + -21.916;
   1:  PR[91,3] = PR[90,3] + 87.501;
   1:L PR[91] R[100]mm/sec CNT100;
   1:  PR[91,1] = PR[90,1] + -40.604;
   1:  PR[91,2] = PR[90,2] + -22.839;
   1:  PR[91,3] = PR[90,3] + 87.521;
   1:L PR[91] R[100]mm/sec CNT100;
   1:  PR[91,1] = PR[90,1] + -37.595;
   1:  PR[91,2] = PR[90,2] + -23.754;
   1:  PR[91,3] = PR[90,3] + 87.531;
   1:L PR[91] R[100]mm/sec CNT100;
   1:  PR[91,1] = PR[90,1] + -34.373;
   1:  PR[91,2] = PR[90,2] + -24.687;
   1:  PR[91,3] = PR[90,3] + 87.545;
   1:L PR[91] R[100]mm/sec CNT100;
   1:  PR[91,1] = PR[90,1] + -31.993;
   1:  PR[91,2] = PR[90,2] + -25.305;
   1:  PR[91,3] = PR[90,3] + 87.559;
   1:L PR[91] R[100]mm/sec CNT100;
   1:  PR[91,1] = PR[90,1] + -22.909;
   1:  PR[91,2] = PR[90,2] + -26.927;
   1:  PR[91,3] = PR[90,3] + 87.570;
   1:L PR[91] R[100]mm/sec CNT100;
   1:  PR[91,1] = PR[90,1] + -19.445;
   1:  PR[91,2] = PR[90,2] + -27.305;
   1:  PR[91,3] = PR[90,3] + 87.609;
   1:L PR[91] R[100]mm/sec CNT100;
   1:  PR[91,1] = PR[90,1] + -13.177;
   1:  PR[91,2] = PR[90,2] + -27.959;
   1:  PR[91,3] = PR[90,3] + 87.624;
   1:L PR[91] R[100]mm/sec CNT100;
   1:  PR[91,1] = PR[90,1] + -6.530;
   1:  PR[91,2] = PR[90,2] + -28.215;
   1:  PR[91,3] = PR[90,3] + 87.651;
   1:L PR[91] R[100]mm/sec CNT100;
   1:  PR[91,1] = PR[90,1] + -2.969;
   1:  PR[91,2] = PR[90,2] + -28.333;
   1:  PR[91,3] = PR[90,3] + 87.679;
   1:L PR[91] R[100]mm/sec CNT100;
   1:  PR[91,1] = PR[90,1] + 7.766;
   1:  PR[91,2] = PR[90,2] + -27.986;
   1:  PR[91,3] = PR[90,3] + 87.694;
   1:L PR[91] R[100]mm/sec CNT100;
   1:  PR[91,1] = PR[90,1] + 9.166;
   1:  PR[91,2] = PR[90,2] + -28.006;
   1:  PR[91,3] = PR[90,3] + 87.740;
   1:L PR[91] R[100]mm/sec CNT100;
   1:  PR[91,1] = PR[90,1] + 10.864;
   1:  PR[91,2] = PR[90,2] + -27.971;
   1:  PR[91,3] = PR[90,3] + 87.746;
   1:L PR[91] R[100]mm/sec CNT100;
   1:  PR[91,1] = PR[90,1] + 12.500;
   1:  PR[91,2] = PR[90,2] + -27.879;
   1:  PR[91,3] = PR[90,3] + 87.753;
   1:L PR[91] R[100]mm/sec CNT100;
   1:  PR[91,1] = PR[90,1] + 13.907;
   1:  PR[91,2] = PR[90,2] + -27.767;
   1:  PR[91,3] = PR[90,3] + 87.760;
   1:L PR[91] R[100]mm/sec CNT100;
   1:  PR[91,1] = PR[90,1] + 17.964;
   1:  PR[91,2] = PR[90,2] + -28.256;
   1:  PR[91,3] = PR[90,3] + 87.766;
   1:L PR[91] R[100]mm/sec CNT100;
   1:  PR[91,1] = PR[90,1] + 18.028;
   1:  PR[91,2] = PR[90,2] + -28.259;
   1:  PR[91,3] = PR[90,3] + 87.784;
   1:L PR[91] R[100]mm/sec CNT100;
   1:  PR[91,1] = PR[90,1] + 23.535;
   1:  PR[91,2] = PR[90,2] + -28.156;
   1:L PR[91] R[100]mm/sec CNT100;
   1:  PR[91,1] = PR[90,1] + 23.597;
   1:  PR[91,2] = PR[90,2] + -28.531;
   1:  PR[91,3] = PR[90,3] + 87.808;
   1:L PR[91] R[100]mm/sec CNT100;
   1:  PR[91,1] = PR[90,1] + 23.842;
   1:  PR[91,2] = PR[90,2] + -28.584;
   1:  PR[91,3] = PR[90,3] + 87.809;
   1:L PR[91] R[100]mm/sec CNT100;
   1:  PR[91,1] = PR[90,1] + 27.676;
   1:  PR[91,2] = PR[90,2] + -29.474;
   1:  PR[91,3] = PR[90,3] + 87.810;
   1:L PR[91] R[100]mm/sec CNT100;
   1:  PR[91,1] = PR[90,1] + 32.886;
   1:  PR[91,2] = PR[90,2] + -29.769;
   1:  PR[91,3] = PR[90,3] + 87.827;
   1:L PR[91] R[100]mm/sec CNT100;
   1:  PR[91,1] = PR[90,1] + 38.004;
   1:  PR[91,2] = PR[90,2] + -29.151;
   1:  PR[91,3] = PR[90,3] + 87.849;
   1:L PR[91] R[100]mm/sec CNT100;
   1:  PR[91,1] = PR[90,1] + 42.904;
   1:  PR[91,2] = PR[90,2] + -27.658;
   1:  PR[91,3] = PR[90,3] + 87.871;
   1:L PR[91] R[100]mm/sec CNT100;
   1:  PR[91,1] = PR[90,1] + 47.549;
   1:  PR[91,2] = PR[90,2] + -25.414;
   1:  PR[91,3] = PR[90,3] + 87.893;
   1:L PR[91] R[100]mm/sec CNT100;
   1:  PR[91,1] = PR[90,1] + 51.641;
   1:  PR[91,2] = PR[90,2] + -22.484;
   1:  PR[91,3] = PR[90,3] + 87.915;
   1:L PR[91] R[100]mm/sec CNT100;
   1:  PR[91,1] = PR[90,1] + 54.090;
   1:  PR[91,2] = PR[90,2] + -19.978;
   1:  PR[91,3] = PR[90,3] + 87.937;
   1:L PR[91] R[100]mm/sec CNT100;
   1:  PR[91,1] = PR[90,1] + 55.118;
   1:  PR[91,2] = PR[90,2] + -19.051;
   1:  PR[91,3] = PR[90,3] + 87.952;
   1:L PR[91] R[100]mm/sec CNT100;
   1:  PR[91,1] = PR[90,1] + 55.443;
   1:  PR[91,2] = PR[90,2] + -18.712;
   1:  PR[91,3] = PR[90,3] + 87.957;
   1:L PR[91] R[100]mm/sec CNT100;
   1:  PR[91,1] = PR[90,1] + 57.489;
   1:  PR[91,2] = PR[90,2] + -16.058;
   1:  PR[91,3] = PR[90,3] + 87.960;
   1:L PR[91] R[100]mm/sec CNT100;
   1:  PR[91,1] = PR[90,1] + 58.739;
   1:  PR[91,2] = PR[90,2] + -14.217;
   1:  PR[91,3] = PR[90,3] + 87.974;
   1:L PR[91] R[100]mm/sec CNT100;
   1:  PR[91,1] = PR[90,1] + 59.321;
   1:  PR[91,2] = PR[90,2] + -13.077;
   1:  PR[91,3] = PR[90,3] + 87.983;
   1:L PR[91] R[100]mm/sec CNT100;
   1:  PR[91,1] = PR[90,1] + 60.647;
   1:  PR[91,2] = PR[90,2] + -10.162;
   1:  PR[91,3] = PR[90,3] + 87.989;
   1:L PR[91] R[100]mm/sec CNT100;
   1:  PR[91,1] = PR[90,1] + 60.947;
   1:  PR[91,2] = PR[90,2] + -9.626;
   1:  PR[91,3] = PR[90,3] + 88.002;
   1:L PR[91] R[100]mm/sec CNT100;
   1:  PR[91,1] = PR[90,1] + 60.967;
   1:  PR[91,2] = PR[90,2] + -9.586;
   1:  PR[91,3] = PR[90,3] + 88.005;
   1:L PR[91] R[100]mm/sec CNT100;
   1:  PR[91,1] = PR[90,1] + 62.074;
   1:  PR[91,2] = PR[90,2] + -6.140;
   1:L PR[91] R[100]mm/sec CNT100;
   1:  PR[91,1] = PR[90,1] + 62.374;
   1:  PR[91,2] = PR[90,2] + -5.080;
   1:  PR[91,3] = PR[90,3] + 88.021;
   1:L PR[91] R[100]mm/sec CNT100;
   1:  PR[91,1] = PR[90,1] + 62.812;
   1:  PR[91,2] = PR[90,2] + -0.723;
   1:  PR[91,3] = PR[90,3] + 88.025;
   1:L PR[91] R[100]mm/sec CNT100;
   1:  PR[91,1] = PR[90,1] + 62.655;
   1:  PR[91,2] = PR[90,2] + 0.936;
   1:  PR[91,3] = PR[90,3] + 88.044;
   1:L PR[91] R[100]mm/sec CNT100;
   1:  PR[91,1] = PR[90,1] + 62.375;
   1:  PR[91,2] = PR[90,2] + 3.618;
   1:  PR[91,3] = PR[90,3] + 88.051;
   1:L PR[91] R[100]mm/sec CNT100;
   1:  PR[91,1] = PR[90,1] + 62.074;
   1:  PR[91,2] = PR[90,2] + 4.681;
   1:  PR[91,3] = PR[90,3] + 88.063;
   1:L PR[91] R[100]mm/sec CNT100;
   1:  PR[91,1] = PR[90,1] + 60.967;
   1:  PR[91,2] = PR[90,2] + 8.127;
   1:  PR[91,3] = PR[90,3] + 88.067;
   1:L PR[91] R[100]mm/sec CNT100;
   1:  PR[91,1] = PR[90,1] + 60.947;
   1:  PR[91,2] = PR[90,2] + 8.167;
   1:  PR[91,3] = PR[90,3] + 88.083;
   1:L PR[91] R[100]mm/sec CNT100;
   1:  PR[91,1] = PR[90,1] + 60.647;
   1:  PR[91,2] = PR[90,2] + 8.703;
   1:L PR[91] R[100]mm/sec CNT100;
   1:  PR[91,1] = PR[90,1] + 59.321;
   1:  PR[91,2] = PR[90,2] + 11.618;
   1:  PR[91,3] = PR[90,3] + 88.086;
   1:L PR[91] R[100]mm/sec CNT100;
   1:  PR[91,1] = PR[90,1] + 58.739;
   1:  PR[91,2] = PR[90,2] + 12.758;
   1:  PR[91,3] = PR[90,3] + 88.099;
   1:L PR[91] R[100]mm/sec CNT100;
   1:  PR[91,1] = PR[90,1] + 57.489;
   1:  PR[91,2] = PR[90,2] + 14.600;
   1:  PR[91,3] = PR[90,3] + 88.105;
   1:L PR[91] R[100]mm/sec CNT100;
   1:  PR[91,1] = PR[90,1] + 55.443;
   1:  PR[91,2] = PR[90,2] + 17.253;
   1:  PR[91,3] = PR[90,3] + 88.114;
   1:L PR[91] R[100]mm/sec CNT100;
   1:  PR[91,1] = PR[90,1] + 55.118;
   1:  PR[91,2] = PR[90,2] + 17.592;
   1:  PR[91,3] = PR[90,3] + 88.129;
   1:L PR[91] R[100]mm/sec CNT100;
   1:  PR[91,1] = PR[90,1] + 54.090;
   1:  PR[91,2] = PR[90,2] + 18.519;
   1:  PR[91,3] = PR[90,3] + 88.131;
   1:L PR[91] R[100]mm/sec CNT100;
   1:  PR[91,1] = PR[90,1] + 51.641;
   1:  PR[91,2] = PR[90,2] + 21.026;
   1:  PR[91,3] = PR[90,3] + 88.136;
   1:L PR[91] R[100]mm/sec CNT100;
   1:  PR[91,1] = PR[90,1] + 47.549;
   1:  PR[91,2] = PR[90,2] + 23.955;
   1:  PR[91,3] = PR[90,3] + 88.151;
   1:L PR[91] R[100]mm/sec CNT100;
   1:  PR[91,1] = PR[90,1] + 42.904;
   1:  PR[91,2] = PR[90,2] + 26.199;
   1:  PR[91,3] = PR[90,3] + 88.173;
   1:L PR[91] R[100]mm/sec CNT100;
   1:  PR[91,1] = PR[90,1] + 38.004;
   1:  PR[91,2] = PR[90,2] + 27.692;
   1:  PR[91,3] = PR[90,3] + 88.195;
   1:L PR[91] R[100]mm/sec CNT100;
   1:  PR[91,1] = PR[90,1] + 32.886;
   1:  PR[91,2] = PR[90,2] + 28.310;
   1:  PR[91,3] = PR[90,3] + 88.217;
   1:L PR[91] R[100]mm/sec CNT100;
   1:  PR[91,1] = PR[90,1] + 27.676;
   1:  PR[91,2] = PR[90,2] + 28.015;
   1:  PR[91,3] = PR[90,3] + 88.239;
   1:L PR[91] R[100]mm/sec CNT100;
   1:  PR[91,1] = PR[90,1] + 23.842;
   1:  PR[91,2] = PR[90,2] + 27.125;
   1:  PR[91,3] = PR[90,3] + 88.261;
   1:L PR[91] R[100]mm/sec CNT100;
   1:  PR[91,1] = PR[90,1] + 22.019;
   1:  PR[91,2] = PR[90,2] + 26.732;
   1:  PR[91,3] = PR[90,3] + 88.278;
   1:L PR[91] R[100]mm/sec CNT100;
   1:  PR[91,1] = PR[90,1] + 18.496;
   1:  PR[91,2] = PR[90,2] + 26.796;
   1:  PR[91,3] = PR[90,3] + 88.286;
   1:L PR[91] R[100]mm/sec CNT100;
   1:  PR[91,1] = PR[90,1] + 17.924;
   1:  PR[91,2] = PR[90,2] + 26.793;
   1:  PR[91,3] = PR[90,3] + 88.301;
   1:L PR[91] R[100]mm/sec CNT100;
   1:  PR[91,1] = PR[90,1] + 13.907;
   1:  PR[91,2] = PR[90,2] + 26.308;
   1:  PR[91,3] = PR[90,3] + 88.303;
   1:L PR[91] R[100]mm/sec CNT100;
   1:  PR[91,1] = PR[90,1] + 12.500;
   1:  PR[91,2] = PR[90,2] + 26.420;
   1:  PR[91,3] = PR[90,3] + 88.320;
   1:L PR[91] R[100]mm/sec CNT100;
   1:  PR[91,1] = PR[90,1] + 10.887;
   1:  PR[91,2] = PR[90,2] + 26.511;
   1:  PR[91,3] = PR[90,3] + 88.326;
   1:L PR[91] R[100]mm/sec CNT100;
   1:  PR[91,1] = PR[90,1] + 8.242;
   1:  PR[91,2] = PR[90,2] + 26.490;
   1:  PR[91,3] = PR[90,3] + 88.333;
   1:L PR[91] R[100]mm/sec CNT100;
   1:  PR[91,1] = PR[90,1] + 6.900;
   1:  PR[91,2] = PR[90,2] + 26.563;
   1:  PR[91,3] = PR[90,3] + 88.345;
   1:L PR[91] R[100]mm/sec CNT100;
   1:  PR[91,1] = PR[90,1] + -2.968;
   1:  PR[91,2] = PR[90,2] + 26.874;
   1:  PR[91,3] = PR[90,3] + 88.350;
   1:L PR[91] R[100]mm/sec CNT100;
   1:  PR[91,1] = PR[90,1] + -6.530;
   1:  PR[91,2] = PR[90,2] + 26.756;
   1:  PR[91,3] = PR[90,3] + 88.392;
   1:L PR[91] R[100]mm/sec CNT100;
   1:  PR[91,1] = PR[90,1] + -13.177;
   1:  PR[91,2] = PR[90,2] + 26.500;
   1:  PR[91,3] = PR[90,3] + 88.408;
   1:L PR[91] R[100]mm/sec CNT100;
   1:  PR[91,1] = PR[90,1] + -19.445;
   1:  PR[91,2] = PR[90,2] + 25.846;
   1:  PR[91,3] = PR[90,3] + 88.436;
   1:L PR[91] R[100]mm/sec CNT100;
   1:  PR[91,1] = PR[90,1] + -22.909;
   1:  PR[91,2] = PR[90,2] + 25.468;
   1:  PR[91,3] = PR[90,3] + 88.463;
   1:L PR[91] R[100]mm/sec CNT100;
   1:  PR[91,1] = PR[90,1] + -31.993;
   1:  PR[91,2] = PR[90,2] + 23.847;
   1:  PR[91,3] = PR[90,3] + 88.478;
   1:L PR[91] R[100]mm/sec CNT100;
   1:  PR[91,1] = PR[90,1] + -34.366;
   1:  PR[91,2] = PR[90,2] + 23.230;
   1:  PR[91,3] = PR[90,3] + 88.517;
   1:L PR[91] R[100]mm/sec CNT100;
   1:  PR[91,1] = PR[90,1] + -41.010;
   1:  PR[91,2] = PR[90,2] + 21.258;
   1:  PR[91,3] = PR[90,3] + 88.528;
   1:L PR[91] R[100]mm/sec CNT100;
   1:  PR[91,1] = PR[90,1] + -42.927;
   1:  PR[91,2] = PR[90,2] + 20.525;
   1:  PR[91,3] = PR[90,3] + 88.557;
   1:L PR[91] R[100]mm/sec CNT100;
   1:  PR[91,1] = PR[90,1] + -45.770;
   1:  PR[91,2] = PR[90,2] + 19.214;
   1:  PR[91,3] = PR[90,3] + 88.566;
   1:L PR[91] R[100]mm/sec CNT100;
   1:  PR[91,1] = PR[90,1] + -49.044;
   1:  PR[91,2] = PR[90,2] + 17.545;
   1:  PR[91,3] = PR[90,3] + 88.579;
   1:L PR[91] R[100]mm/sec CNT100;
   1:  PR[91] = PR[90];
   1:  PR[91,1] = PR[90,1] + -52.926;
   1:  PR[91,2] = PR[90,2] + 13.640;
   1:  PR[91,3] = PR[90,3] + 89.895;
   1:L PR[91] R[100]mm/sec CNT100;
   1:  PR[91,1] = PR[90,1] + -56.042;
   1:  PR[91,2] = PR[90,2] + 10.206;
   1:  PR[91,3] = PR[90,3] + 88.619;
   1:L PR[91] R[100]mm/sec CNT100;
   1:  PR[91,1] = PR[90,1] + -56.949;
   1:  PR[91,2] = PR[90,2] + 9.159;
   1:  PR[91,3] = PR[90,3] + 88.639;
   1:L PR[91] R[100]mm/sec CNT100;
   1:  PR[91,1] = PR[90,1] + -59.443;
   1:  PR[91,2] = PR[90,2] + 4.317;
   1:  PR[91,3] = PR[90,3] + 88.645;
   1:L PR[91] R[100]mm/sec CNT100;
   1:  PR[91,1] = PR[90,1] + -59.446;
   1:  PR[91,2] = PR[90,2] + 4.299;
   1:  PR[91,3] = PR[90,3] + 88.668;
   1:L PR[91] R[100]mm/sec CNT100;
   1:  PR[91,1] = PR[90,1] + -60.232;
   1:  PR[91,2] = PR[90,2] + -0.740;
   1:L PR[91] R[100]mm/sec CNT100;
   1:  PR[91,1] = PR[90,1] + -60.086;
   1:  PR[91,2] = PR[90,2] + -1.741;
   1:  PR[91,3] = PR[90,3] + 88.690;
   1:L PR[91] R[100]mm/sec CNT100;
   1:  PR[91,1] = PR[90,1] + -59.602;
   1:  PR[91,2] = PR[90,2] + -4.260;
   1:  PR[91,3] = PR[90,3] + 88.695;
   1:L PR[91] R[100]mm/sec CNT100;
   1:  PR[91,1] = PR[90,1] + -59.526;
   1:  PR[91,2] = PR[90,2] + -4.467;
   1:  PR[91,3] = PR[90,3] + 88.706;
   1:L PR[91] R[100]mm/sec CNT100;
   1:  PR[91,1] = PR[90,1] + -59.377;
   1:  PR[91,2] = PR[90,2] + -5.416;
   1:  PR[91,3] = PR[90,3] + 88.707;
   1:L PR[91] R[100]mm/sec CNT100;
   1:  PR[91,1] = PR[90,1] + -57.834;
   1:  PR[91,2] = PR[90,2] + -8.715;
   1:  PR[91,3] = PR[90,3] + 88.711;
   1:L PR[91] R[100]mm/sec CNT100;
   1:  PR[91,1] = PR[90,1] + -57.168;
   1:  PR[91,2] = PR[90,2] + -10.096;
   1:  PR[91,3] = PR[90,3] + 88.727;
   1:L PR[91] R[100]mm/sec CNT100;
   1:  PR[91,1] = PR[90,1] + -55.257;
   1:  PR[91,2] = PR[90,2] + -12.427;
   1:  PR[91,3] = PR[90,3] + 88.733;
   1:L PR[91] R[100]mm/sec CNT100;
   1:  PR[91,1] = PR[90,1] + -53.331;
   1:  PR[91,2] = PR[90,2] + -14.694;
   1:  PR[91,3] = PR[90,3] + 88.746;
   1:L PR[91] R[100]mm/sec CNT100;
   1:  PR[91,1] = PR[90,1] + -51.908;
   1:  PR[91,2] = PR[90,2] + -15.839;
   1:  PR[91,3] = PR[90,3] + 88.759;
   1:L PR[91] R[100]mm/sec CNT100;
   1:  PR[91,1] = PR[90,1] + -47.806;
   1:  PR[91,2] = PR[90,2] + -18.993;
   1:  PR[91,3] = PR[90,3] + 88.767;
   1:L PR[91] R[100]mm/sec CNT100;
   1:  PR[91,1] = PR[90,1] + -41.701;
   1:  PR[91,2] = PR[90,2] + -21.799;
   1:  PR[91,3] = PR[90,3] + 88.789;
   1:L PR[91] R[100]mm/sec CNT100;
   1:  PR[91,1] = PR[90,1] + -38.057;
   1:  PR[91,2] = PR[90,2] + -23.210;
   1:  PR[91,3] = PR[90,3] + 88.818;
   1:L PR[91] R[100]mm/sec CNT100;
   1:  PR[91,1] = PR[90,1] + -36.603;
   1:  PR[91,2] = PR[90,2] + -23.652;
   1:  PR[91,3] = PR[90,3] + 88.835;
   1:L PR[91] R[100]mm/sec CNT100;
   1:  PR[91,1] = PR[90,1] + -35.021;
   1:  PR[91,2] = PR[90,2] + -24.110;
   1:  PR[91,3] = PR[90,3] + 88.842;
   1:L PR[91] R[100]mm/sec CNT100;
   1:  PR[91,1] = PR[90,1] + -29.592;
   1:  PR[91,2] = PR[90,2] + -25.521;
   1:  PR[91,3] = PR[90,3] + 88.849;
   1:L PR[91] R[100]mm/sec CNT100;
   1:  PR[91,1] = PR[90,1] + -20.438;
   1:  PR[91,2] = PR[90,2] + -27.159;
   1:  PR[91,3] = PR[90,3] + 88.873;
   1:L PR[91] R[100]mm/sec CNT100;
   1:  PR[91,1] = PR[90,1] + -16.033;
   1:  PR[91,2] = PR[90,2] + -27.640;
   1:  PR[91,3] = PR[90,3] + 88.913;
   1:L PR[91] R[100]mm/sec CNT100;
   1:  PR[91,1] = PR[90,1] + -10.631;
   1:  PR[91,2] = PR[90,2] + -28.203;
   1:  PR[91,3] = PR[90,3] + 88.932;
   1:L PR[91] R[100]mm/sec CNT100;
   1:  PR[91,1] = PR[90,1] + -2.987;
   1:  PR[91,2] = PR[90,2] + -28.498;
   1:  PR[91,3] = PR[90,3] + 88.956;
   1:L PR[91] R[100]mm/sec CNT100;
   1:  PR[91,1] = PR[90,1] + -0.342;
   1:  PR[91,2] = PR[90,2] + -28.586;
   1:  PR[91,3] = PR[90,3] + 88.989;
   1:L PR[91] R[100]mm/sec CNT100;
   1:  PR[91,1] = PR[90,1] + 9.329;
   1:  PR[91,2] = PR[90,2] + -28.281;
   1:  PR[91,3] = PR[90,3] + 89.000;
   1:L PR[91] R[100]mm/sec CNT100;
   1:  PR[91,1] = PR[90,1] + 10.609;
   1:  PR[91,2] = PR[90,2] + -28.228;
   1:  PR[91,3] = PR[90,3] + 89.042;
   1:L PR[91] R[100]mm/sec CNT100;
   1:  PR[91,1] = PR[90,1] + 11.898;
   1:  PR[91,2] = PR[90,2] + -28.202;
   1:  PR[91,3] = PR[90,3] + 89.047;
   1:L PR[91] R[100]mm/sec CNT100;
   1:  PR[91,1] = PR[90,1] + 13.967;
   1:  PR[91,2] = PR[90,2] + -28.086;
   1:  PR[91,3] = PR[90,3] + 89.053;
   1:L PR[91] R[100]mm/sec CNT100;
   1:  PR[91,1] = PR[90,1] + 14.757;
   1:  PR[91,2] = PR[90,2] + -28.023;
   1:  PR[91,3] = PR[90,3] + 89.062;
   1:L PR[91] R[100]mm/sec CNT100;
   1:  PR[91,1] = PR[90,1] + 16.691;
   1:  PR[91,2] = PR[90,2] + -28.260;
   1:  PR[91,3] = PR[90,3] + 89.065;
   1:L PR[91] R[100]mm/sec CNT100;
   1:  PR[91,1] = PR[90,1] + 18.052;
   1:  PR[91,2] = PR[90,2] + -28.399;
   1:  PR[91,3] = PR[90,3] + 89.074;
   1:L PR[91] R[100]mm/sec CNT100;
   1:  PR[91,1] = PR[90,1] + 18.662;
   1:  PR[91,2] = PR[90,2] + -28.427;
   1:  PR[91,3] = PR[90,3] + 89.079;
   1:L PR[91] R[100]mm/sec CNT100;
   1:  PR[91,1] = PR[90,1] + 23.335;
   1:  PR[91,2] = PR[90,2] + -28.340;
   1:  PR[91,3] = PR[90,3] + 89.082;
   1:L PR[91] R[100]mm/sec CNT100;
   1:  PR[91,1] = PR[90,1] + 23.411;
   1:  PR[91,2] = PR[90,2] + -28.745;
   1:  PR[91,3] = PR[90,3] + 89.102;
   1:L PR[91] R[100]mm/sec CNT100;
   1:  PR[91,1] = PR[90,1] + 27.421;
   1:  PR[91,2] = PR[90,2] + -29.668;
   1:  PR[91,3] = PR[90,3] + 89.104;
   1:L PR[91] R[100]mm/sec CNT100;
   1:  PR[91,1] = PR[90,1] + 32.665;
   1:  PR[91,2] = PR[90,2] + -29.960;
   1:  PR[91,3] = PR[90,3] + 89.122;
   1:L PR[91] R[100]mm/sec CNT100;
   1:  PR[91,1] = PR[90,1] + 37.819;
   1:  PR[91,2] = PR[90,2] + -29.339;
   1:  PR[91,3] = PR[90,3] + 89.144;
   1:L PR[91] R[100]mm/sec CNT100;
   1:  PR[91,1] = PR[90,1] + 42.716;
   1:  PR[91,2] = PR[90,2] + -27.843;
   1:  PR[91,3] = PR[90,3] + 89.167;
   1:L PR[91] R[100]mm/sec CNT100;
   1:  PR[91,1] = PR[90,1] + 45.674;
   1:  PR[91,2] = PR[90,2] + -26.321;
   1:  PR[91,3] = PR[90,3] + 89.189;
   1:L PR[91] R[100]mm/sec CNT100;
   1:  PR[91,1] = PR[90,1] + 47.308;
   1:  PR[91,2] = PR[90,2] + -25.531;
   1:  PR[91,3] = PR[90,3] + 89.203;
   1:L PR[91] R[100]mm/sec CNT100;
   1:  PR[91,1] = PR[90,1] + 51.432;
   1:  PR[91,2] = PR[90,2] + -22.575;
   1:  PR[91,3] = PR[90,3] + 89.211;
   1:L PR[91] R[100]mm/sec CNT100;
   1:  PR[91,1] = PR[90,1] + 54.911;
   1:  PR[91,2] = PR[90,2] + -19.016;
   1:  PR[91,3] = PR[90,3] + 89.233;
   1:L PR[91] R[100]mm/sec CNT100;
   1:  PR[91,1] = PR[90,1] + 56.172;
   1:  PR[91,2] = PR[90,2] + -17.160;
   1:  PR[91,3] = PR[90,3] + 89.254;
   1:L PR[91] R[100]mm/sec CNT100;
   1:  PR[91,1] = PR[90,1] + 57.617;
   1:  PR[91,2] = PR[90,2] + -15.286;
   1:  PR[91,3] = PR[90,3] + 89.264;
   1:L PR[91] R[100]mm/sec CNT100;
   1:  PR[91,1] = PR[90,1] + 58.051;
   1:  PR[91,2] = PR[90,2] + -14.646;
   1:  PR[91,3] = PR[90,3] + 89.274;
   1:L PR[91] R[100]mm/sec CNT100;
   1:  PR[91,1] = PR[90,1] + 59.413;
   1:  PR[91,2] = PR[90,2] + -11.978;
   1:  PR[91,3] = PR[90,3] + 89.278;
   1:L PR[91] R[100]mm/sec CNT100;
   1:  PR[91,1] = PR[90,1] + 60.325;
   1:  PR[91,2] = PR[90,2] + -9.973;
   1:  PR[91,3] = PR[90,3] + 89.291;
   1:L PR[91] R[100]mm/sec CNT100;
   1:  PR[91,1] = PR[90,1] + 60.726;
   1:  PR[91,2] = PR[90,2] + -8.594;
   1:  PR[91,3] = PR[90,3] + 89.300;
   1:L PR[91] R[100]mm/sec CNT100;
   1:  PR[91,1] = PR[90,1] + 61.580;
   1:  PR[91,2] = PR[90,2] + -5.335;
   1:  PR[91,3] = PR[90,3] + 89.306;
   1:L PR[91] R[100]mm/sec CNT100;
   1:  PR[91,1] = PR[90,1] + 61.980;
   1:  PR[91,2] = PR[90,2] + -0.770;
   1:  PR[91,3] = PR[90,3] + 89.321;
   1:L PR[91] R[100]mm/sec CNT100;
   1:  PR[91,1] = PR[90,1] + 61.703;
   1:  PR[91,2] = PR[90,2] + 2.215;
   1:  PR[91,3] = PR[90,3] + 89.341;
   1:L PR[91] R[100]mm/sec CNT100;
   1:  PR[91,1] = PR[90,1] + 61.577;
   1:  PR[91,2] = PR[90,2] + 3.888;
   1:  PR[91,3] = PR[90,3] + 89.354;
   1:L PR[91] R[100]mm/sec CNT100;
   1:  PR[91,1] = PR[90,1] + 60.726;
   1:  PR[91,2] = PR[90,2] + 7.135;
   1:  PR[91,3] = PR[90,3] + 89.361;
   1:L PR[91] R[100]mm/sec CNT100;
   1:  PR[91,1] = PR[90,1] + 60.325;
   1:  PR[91,2] = PR[90,2] + 8.514;
   1:  PR[91,3] = PR[90,3] + 89.375;
   1:L PR[91] R[100]mm/sec CNT100;
   1:  PR[91,1] = PR[90,1] + 59.413;
   1:  PR[91,2] = PR[90,2] + 10.519;
   1:  PR[91,3] = PR[90,3] + 89.381;
   1:L PR[91] R[100]mm/sec CNT100;
   1:  PR[91,1] = PR[90,1] + 58.051;
   1:  PR[91,2] = PR[90,2] + 13.187;
   1:  PR[91,3] = PR[90,3] + 89.391;
   1:L PR[91] R[100]mm/sec CNT100;
   1:  PR[91,1] = PR[90,1] + 57.617;
   1:  PR[91,2] = PR[90,2] + 13.827;
   1:  PR[91,3] = PR[90,3] + 89.404;
   1:L PR[91] R[100]mm/sec CNT100;
   1:  PR[91,1] = PR[90,1] + 56.172;
   1:  PR[91,2] = PR[90,2] + 15.701;
   1:  PR[91,3] = PR[90,3] + 89.407;
   1:L PR[91] R[100]mm/sec CNT100;
   1:  PR[91,1] = PR[90,1] + 54.911;
   1:  PR[91,2] = PR[90,2] + 17.557;
   1:  PR[91,3] = PR[90,3] + 89.417;
   1:L PR[91] R[100]mm/sec CNT100;
   1:  PR[91,1] = PR[90,1] + 51.432;
   1:  PR[91,2] = PR[90,2] + 21.116;
   1:  PR[91,3] = PR[90,3] + 89.427;
   1:L PR[91] R[100]mm/sec CNT100;
   1:  PR[91,1] = PR[90,1] + 47.308;
   1:  PR[91,2] = PR[90,2] + 24.072;
   1:  PR[91,3] = PR[90,3] + 89.449;
   1:L PR[91] R[100]mm/sec CNT100;
   1:  PR[91,1] = PR[90,1] + 45.674;
   1:  PR[91,2] = PR[90,2] + 24.862;
   1:  PR[91,3] = PR[90,3] + 89.470;
   1:L PR[91] R[100]mm/sec CNT100;
   1:  PR[91,1] = PR[90,1] + 42.716;
   1:  PR[91,2] = PR[90,2] + 26.384;
   1:  PR[91,3] = PR[90,3] + 89.478;
   1:L PR[91] R[100]mm/sec CNT100;
   1:  PR[91,1] = PR[90,1] + 37.819;
   1:  PR[91,2] = PR[90,2] + 27.880;
   1:  PR[91,3] = PR[90,3] + 89.493;
   1:L PR[91] R[100]mm/sec CNT100;
   1:  PR[91,1] = PR[90,1] + 32.665;
   1:  PR[91,2] = PR[90,2] + 28.501;
   1:  PR[91,3] = PR[90,3] + 89.515;
   1:L PR[91] R[100]mm/sec CNT100;
   1:  PR[91,1] = PR[90,1] + 27.421;
   1:  PR[91,2] = PR[90,2] + 28.210;
   1:  PR[91,3] = PR[90,3] + 89.537;
   1:L PR[91] R[100]mm/sec CNT100;
   1:  PR[91,1] = PR[90,1] + 21.849;
   1:  PR[91,2] = PR[90,2] + 26.926;
   1:  PR[91,3] = PR[90,3] + 89.560;
   1:L PR[91] R[100]mm/sec CNT100;
   1:  PR[91,1] = PR[90,1] + 18.668;
   1:  PR[91,2] = PR[90,2] + 26.969;
   1:  PR[91,3] = PR[90,3] + 89.584;
   1:L PR[91] R[100]mm/sec CNT100;
   1:  PR[91,1] = PR[90,1] + 18.073;
   1:  PR[91,2] = PR[90,2] + 26.941;
   1:  PR[91,3] = PR[90,3] + 89.598;
   1:L PR[91] R[100]mm/sec CNT100;
   1:  PR[91,1] = PR[90,1] + 15.356;
   1:  PR[91,2] = PR[90,2] + 26.609;
   1:  PR[91,3] = PR[90,3] + 89.601;
   1:L PR[91] R[100]mm/sec CNT100;
   1:  PR[91,1] = PR[90,1] + 14.693;
   1:  PR[91,2] = PR[90,2] + 26.569;
   1:  PR[91,3] = PR[90,3] + 89.612;
   1:L PR[91] R[100]mm/sec CNT100;
   1:  PR[91,1] = PR[90,1] + 13.967;
   1:  PR[91,2] = PR[90,2] + 26.627;
   1:  PR[91,3] = PR[90,3] + 89.615;
   1:L PR[91] R[100]mm/sec CNT100;
   1:  PR[91,1] = PR[90,1] + 11.919;
   1:  PR[91,2] = PR[90,2] + 26.742;
   1:  PR[91,3] = PR[90,3] + 89.619;
   1:L PR[91] R[100]mm/sec CNT100;
   1:  PR[91,1] = PR[90,1] + 11.052;
   1:  PR[91,2] = PR[90,2] + 26.735;
   1:  PR[91,3] = PR[90,3] + 89.627;
   1:L PR[91] R[100]mm/sec CNT100;
   1:  PR[91,1] = PR[90,1] + 10.556;
   1:  PR[91,2] = PR[90,2] + 26.772;
   1:  PR[91,3] = PR[90,3] + 89.631;
   1:L PR[91] R[100]mm/sec CNT100;
   1:  PR[91,1] = PR[90,1] + 9.329;
   1:  PR[91,2] = PR[90,2] + 26.822;
   1:  PR[91,3] = PR[90,3] + 89.633;
   1:L PR[91] R[100]mm/sec CNT100;
   1:  PR[91,1] = PR[90,1] + -0.341;
   1:  PR[91,2] = PR[90,2] + 27.127;
   1:  PR[91,3] = PR[90,3] + 89.639;
   1:L PR[91] R[100]mm/sec CNT100;
   1:  PR[91,1] = PR[90,1] + -2.989;
   1:  PR[91,2] = PR[90,2] + 27.039;
   1:  PR[91,3] = PR[90,3] + 89.680;
   1:L PR[91] R[100]mm/sec CNT100;
   1:  PR[91,1] = PR[90,1] + -10.631;
   1:  PR[91,2] = PR[90,2] + 26.744;
   1:  PR[91,3] = PR[90,3] + 89.692;
   1:L PR[91] R[100]mm/sec CNT100;
   1:  PR[91,1] = PR[90,1] + -16.033;
   1:  PR[91,2] = PR[90,2] + 26.181;
   1:  PR[91,3] = PR[90,3] + 89.725;
   1:L PR[91] R[100]mm/sec CNT100;
   1:  PR[91,1] = PR[90,1] + -20.438;
   1:  PR[91,2] = PR[90,2] + 25.700;
   1:  PR[91,3] = PR[90,3] + 89.748;
   1:L PR[91] R[100]mm/sec CNT100;
   1:  PR[91,1] = PR[90,1] + -29.592;
   1:  PR[91,2] = PR[90,2] + 24.062;
   1:  PR[91,3] = PR[90,3] + 89.767;
   1:L PR[91] R[100]mm/sec CNT100;
   1:  PR[91,1] = PR[90,1] + -35.015;
   1:  PR[91,2] = PR[90,2] + 22.653;
   1:  PR[91,3] = PR[90,3] + 89.807;
   1:L PR[91] R[100]mm/sec CNT100;
   1:  PR[91,1] = PR[90,1] + -38.264;
   1:  PR[91,2] = PR[90,2] + 21.688;
   1:  PR[91,3] = PR[90,3] + 89.832;
   1:L PR[91] R[100]mm/sec CNT100;
   1:  PR[91,1] = PR[90,1] + -41.654;
   1:  PR[91,2] = PR[90,2] + 20.393;
   1:  PR[91,3] = PR[90,3] + 89.846;
   1:L PR[91] R[100]mm/sec CNT100;
   1:  PR[91,1] = PR[90,1] + -46.607;
   1:  PR[91,2] = PR[90,2] + 18.108;
   1:  PR[91,3] = PR[90,3] + 89.862;
   1:L PR[91] R[100]mm/sec CNT100;
   1:  PR[91,1] = PR[90,1] + -47.701;
   1:  PR[91,2] = PR[90,2] + 17.551;
   1:  PR[91,3] = PR[90,3] + 89.885;
   1:L PR[91] R[100]mm/sec CNT100;
   1:  PR[91,1] = PR[90,1] + -48.527;
   1:  PR[91,2] = PR[90,2] + 16.958;
   1:  PR[91,3] = PR[90,3] + 89.891;
   1:L PR[91] R[100]mm/sec CNT100;
   1:  PR[91] = PR[90];
   1:  PR[91,1] = PR[90,1] + -51.523;
   1:  PR[91,2] = PR[90,2] + 13.631;
   1:  PR[91,3] = PR[90,3] + 91.195;
   1:L PR[91] R[100]mm/sec CNT100;
   1:  PR[91,1] = PR[90,1] + -53.566;
   1:  PR[91,2] = PR[90,2] + 11.379;
   1:  PR[91,3] = PR[90,3] + 89.919;
   1:L PR[91] R[100]mm/sec CNT100;
   1:  PR[91,1] = PR[90,1] + -55.500;
   1:  PR[91,2] = PR[90,2] + 9.146;
   1:  PR[91,3] = PR[90,3] + 89.932;
   1:L PR[91] R[100]mm/sec CNT100;
   1:  PR[91,1] = PR[90,1] + -57.602;
   1:  PR[91,2] = PR[90,2] + 5.064;
   1:  PR[91,3] = PR[90,3] + 89.945;
   1:L PR[91] R[100]mm/sec CNT100;
   1:  PR[91,1] = PR[90,1] + -57.980;
   1:  PR[91,2] = PR[90,2] + 4.293;
   1:  PR[91,3] = PR[90,3] + 89.965;
   1:L PR[91] R[100]mm/sec CNT100;
   1:  PR[91,1] = PR[90,1] + -58.798;
   1:  PR[91,2] = PR[90,2] + -0.549;
   1:  PR[91,3] = PR[90,3] + 89.969;
   1:L PR[91] R[100]mm/sec CNT100;
   1:  PR[91,1] = PR[90,1] + -58.839;
   1:  PR[91,2] = PR[90,2] + -0.745;
   1:  PR[91,3] = PR[90,3] + 89.990;
   1:L PR[91] R[100]mm/sec CNT100;
   1:  PR[91,1] = PR[90,1] + -58.330;
   1:  PR[91,2] = PR[90,2] + -3.391;
   1:  PR[91,3] = PR[90,3] + 89.991;
   1:L PR[91] R[100]mm/sec CNT100;
   1:  PR[91,1] = PR[90,1] + -58.204;
   1:  PR[91,2] = PR[90,2] + -3.732;
   1:  PR[91,3] = PR[90,3] + 90.003;
   1:L PR[91] R[100]mm/sec CNT100;
   1:  PR[91,1] = PR[90,1] + -57.931;
   1:  PR[91,2] = PR[90,2] + -5.477;
   1:  PR[91,3] = PR[90,3] + 90.004;
   1:L PR[91] R[100]mm/sec CNT100;
   1:  PR[91,1] = PR[90,1] + -56.698;
   1:  PR[91,2] = PR[90,2] + -8.113;
   1:  PR[91,3] = PR[90,3] + 90.012;
   1:L PR[91] R[100]mm/sec CNT100;
   1:  PR[91,1] = PR[90,1] + -55.683;
   1:  PR[91,2] = PR[90,2] + -10.216;
   1:  PR[91,3] = PR[90,3] + 90.025;
   1:L PR[91] R[100]mm/sec CNT100;
   1:  PR[91,1] = PR[90,1] + -54.260;
   1:  PR[91,2] = PR[90,2] + -11.952;
   1:  PR[91,3] = PR[90,3] + 90.035;
   1:L PR[91] R[100]mm/sec CNT100;
   1:  PR[91,1] = PR[90,1] + -51.781;
   1:  PR[91,2] = PR[90,2] + -14.870;
   1:  PR[91,3] = PR[90,3] + 90.045;
   1:L PR[91] R[100]mm/sec CNT100;
   1:  PR[91,1] = PR[90,1] + -51.015;
   1:  PR[91,2] = PR[90,2] + -15.487;
   1:  PR[91,3] = PR[90,3] + 90.061;
   1:L PR[91] R[100]mm/sec CNT100;
   1:  PR[91,1] = PR[90,1] + -48.599;
   1:  PR[91,2] = PR[90,2] + -17.345;
   1:  PR[91,3] = PR[90,3] + 90.066;
   1:L PR[91] R[100]mm/sec CNT100;
   1:  PR[91,1] = PR[90,1] + -46.209;
   1:  PR[91,2] = PR[90,2] + -18.944;
   1:  PR[91,3] = PR[90,3] + 90.079;
   1:L PR[91] R[100]mm/sec CNT100;
   1:  PR[91,1] = PR[90,1] + -44.861;
   1:  PR[91,2] = PR[90,2] + -19.639;
   1:  PR[91,3] = PR[90,3] + 90.092;
   1:L PR[91] R[100]mm/sec CNT100;
   1:  PR[91,1] = PR[90,1] + -40.414;
   1:  PR[91,2] = PR[90,2] + -21.682;
   1:  PR[91,3] = PR[90,3] + 90.098;
   1:L PR[91] R[100]mm/sec CNT100;
   1:  PR[91,1] = PR[90,1] + -35.551;
   1:  PR[91,2] = PR[90,2] + -23.564;
   1:  PR[91,3] = PR[90,3] + 90.119;
   1:L PR[91] R[100]mm/sec CNT100;
   1:  PR[91,1] = PR[90,1] + -27.190;
   1:  PR[91,2] = PR[90,2] + -25.737;
   1:  PR[91,3] = PR[90,3] + 90.142;
   1:L PR[91] R[100]mm/sec CNT100;
   1:  PR[91,1] = PR[90,1] + -17.967;
   1:  PR[91,2] = PR[90,2] + -27.391;
   1:  PR[91,3] = PR[90,3] + 90.180;
   1:L PR[91] R[100]mm/sec CNT100;
   1:  PR[91,1] = PR[90,1] + -12.621;
   1:  PR[91,2] = PR[90,2] + -27.975;
   1:  PR[91,3] = PR[90,3] + 90.221;
   1:L PR[91] R[100]mm/sec CNT100;
   1:  PR[91,1] = PR[90,1] + -8.086;
   1:  PR[91,2] = PR[90,2] + -28.448;
   1:  PR[91,3] = PR[90,3] + 90.244;
   1:L PR[91] R[100]mm/sec CNT100;
   1:  PR[91,1] = PR[90,1] + 2.289;
   1:  PR[91,2] = PR[90,2] + -28.838;
   1:  PR[91,3] = PR[90,3] + 90.264;
   1:L PR[91] R[100]mm/sec CNT100;
   1:  PR[91,1] = PR[90,1] + 10.823;
   1:  PR[91,2] = PR[90,2] + -28.561;
   1:  PR[91,3] = PR[90,3] + 90.309;
   1:L PR[91] R[100]mm/sec CNT100;
   1:  PR[91,1] = PR[90,1] + 13.810;
   1:  PR[91,2] = PR[90,2] + -28.429;
   1:  PR[91,3] = PR[90,3] + 90.347;
   1:L PR[91] R[100]mm/sec CNT100;
   1:  PR[91,1] = PR[90,1] + 15.592;
   1:  PR[91,2] = PR[90,2] + -28.281;
   1:  PR[91,3] = PR[90,3] + 90.360;
   1:L PR[91] R[100]mm/sec CNT100;
   1:  PR[91,1] = PR[90,1] + 18.160;
   1:  PR[91,2] = PR[90,2] + -28.542;
   1:  PR[91,3] = PR[90,3] + 90.367;
   1:L PR[91] R[100]mm/sec CNT100;
   1:  PR[91,1] = PR[90,1] + 19.296;
   1:  PR[91,2] = PR[90,2] + -28.595;
   1:  PR[91,3] = PR[90,3] + 90.379;
   1:L PR[91] R[100]mm/sec CNT100;
   1:  PR[91,1] = PR[90,1] + 23.157;
   1:  PR[91,2] = PR[90,2] + -28.523;
   1:  PR[91,3] = PR[90,3] + 90.384;
   1:L PR[91] R[100]mm/sec CNT100;
   1:  PR[91,1] = PR[90,1] + 23.238;
   1:  PR[91,2] = PR[90,2] + -28.935;
   1:  PR[91,3] = PR[90,3] + 90.400;
   1:L PR[91] R[100]mm/sec CNT100;
   1:  PR[91,1] = PR[90,1] + 27.173;
   1:  PR[91,2] = PR[90,2] + -29.863;
   1:  PR[91,3] = PR[90,3] + 90.402;
   1:L PR[91] R[100]mm/sec CNT100;
   1:  PR[91,1] = PR[90,1] + 32.444;
   1:  PR[91,2] = PR[90,2] + -30.151;
   1:  PR[91,3] = PR[90,3] + 90.420;
   1:L PR[91] R[100]mm/sec CNT100;
   1:  PR[91,1] = PR[90,1] + 37.636;
   1:  PR[91,2] = PR[90,2] + -29.526;
   1:  PR[91,3] = PR[90,3] + 90.443;
   1:L PR[91] R[100]mm/sec CNT100;
   1:  PR[91,1] = PR[90,1] + 42.574;
   1:  PR[91,2] = PR[90,2] + -28.024;
   1:  PR[91,3] = PR[90,3] + 90.466;
   1:L PR[91] R[100]mm/sec CNT100;
   1:  PR[91,1] = PR[90,1] + 47.097;
   1:  PR[91,2] = PR[90,2] + -25.706;
   1:  PR[91,3] = PR[90,3] + 90.488;
   1:L PR[91] R[100]mm/sec CNT100;
   1:  PR[91,1] = PR[90,1] + 48.892;
   1:  PR[91,2] = PR[90,2] + -24.337;
   1:  PR[91,3] = PR[90,3] + 90.510;
   1:L PR[91] R[100]mm/sec CNT100;
   1:  PR[91,1] = PR[90,1] + 51.223;
   1:  PR[91,2] = PR[90,2] + -22.665;
   1:  PR[91,3] = PR[90,3] + 90.520;
   1:L PR[91] R[100]mm/sec CNT100;
   1:  PR[91,1] = PR[90,1] + 54.732;
   1:  PR[91,2] = PR[90,2] + -19.081;
   1:  PR[91,3] = PR[90,3] + 90.533;
   1:L PR[91] R[100]mm/sec CNT100;
   1:  PR[91,1] = PR[90,1] + 57.517;
   1:  PR[91,2] = PR[90,2] + -14.985;
   1:  PR[91,3] = PR[90,3] + 90.555;
   1:L PR[91] R[100]mm/sec CNT100;
   1:  PR[91,1] = PR[90,1] + 58.305;
   1:  PR[91,2] = PR[90,2] + -13.230;
   1:  PR[91,3] = PR[90,3] + 90.576;
   1:L PR[91] R[100]mm/sec CNT100;
   1:  PR[91,1] = PR[90,1] + 59.505;
   1:  PR[91,2] = PR[90,2] + -10.878;
   1:  PR[91,3] = PR[90,3] + 90.585;
   1:L PR[91] R[100]mm/sec CNT100;
   1:  PR[91,1] = PR[90,1] + 59.774;
   1:  PR[91,2] = PR[90,2] + -10.289;
   1:  PR[91,3] = PR[90,3] + 90.596;
   1:L PR[91] R[100]mm/sec CNT100;
   1:  PR[91,1] = PR[90,1] + 60.701;
   1:  PR[91,2] = PR[90,2] + -7.100;
   1:  PR[91,3] = PR[90,3] + 90.599;
   1:L PR[91] R[100]mm/sec CNT100;
   1:  PR[91,1] = PR[90,1] + 61.119;
   1:  PR[91,2] = PR[90,2] + -5.502;
   1:  PR[91,3] = PR[90,3] + 90.613;
   1:L PR[91] R[100]mm/sec CNT100;
   1:  PR[91,1] = PR[90,1] + 61.319;
   1:  PR[91,2] = PR[90,2] + -3.222;
   1:  PR[91,3] = PR[90,3] + 90.621;
   1:L PR[91] R[100]mm/sec CNT100;
   1:  PR[91,1] = PR[90,1] + 61.346;
   1:  PR[91,2] = PR[90,2] + -2.444;
   1:  PR[91,3] = PR[90,3] + 90.631;
   1:L PR[91] R[100]mm/sec CNT100;
   1:  PR[91,1] = PR[90,1] + 61.506;
   1:  PR[91,2] = PR[90,2] + -0.705;
   1:  PR[91,3] = PR[90,3] + 90.634;
   1:L PR[91] R[100]mm/sec CNT100;
   1:  PR[91,1] = PR[90,1] + 61.354;
   1:  PR[91,2] = PR[90,2] + 1.542;
   1:  PR[91,3] = PR[90,3] + 90.642;
   1:L PR[91] R[100]mm/sec CNT100;
   1:  PR[91,1] = PR[90,1] + 61.121;
   1:  PR[91,2] = PR[90,2] + 4.037;
   1:  PR[91,3] = PR[90,3] + 90.651;
   1:L PR[91] R[100]mm/sec CNT100;
   1:  PR[91,1] = PR[90,1] + 60.700;
   1:  PR[91,2] = PR[90,2] + 5.641;
   1:  PR[91,3] = PR[90,3] + 90.662;
   1:L PR[91] R[100]mm/sec CNT100;
   1:  PR[91,1] = PR[90,1] + 59.774;
   1:  PR[91,2] = PR[90,2] + 8.830;
   1:  PR[91,3] = PR[90,3] + 90.670;
   1:L PR[91] R[100]mm/sec CNT100;
   1:  PR[91,1] = PR[90,1] + 59.505;
   1:  PR[91,2] = PR[90,2] + 9.420;
   1:  PR[91,3] = PR[90,3] + 90.684;
   1:L PR[91] R[100]mm/sec CNT100;
   1:  PR[91,1] = PR[90,1] + 58.305;
   1:  PR[91,2] = PR[90,2] + 11.771;
   1:  PR[91,3] = PR[90,3] + 90.687;
   1:L PR[91] R[100]mm/sec CNT100;
   1:  PR[91,1] = PR[90,1] + 57.517;
   1:  PR[91,2] = PR[90,2] + 13.526;
   1:  PR[91,3] = PR[90,3] + 90.698;
   1:L PR[91] R[100]mm/sec CNT100;
   1:  PR[91,1] = PR[90,1] + 54.732;
   1:  PR[91,2] = PR[90,2] + 17.622;
   1:  PR[91,3] = PR[90,3] + 90.707;
   1:L PR[91] R[100]mm/sec CNT100;
   1:  PR[91,1] = PR[90,1] + 51.223;
   1:  PR[91,2] = PR[90,2] + 21.207;
   1:  PR[91,3] = PR[90,3] + 90.728;
   1:L PR[91] R[100]mm/sec CNT100;
   1:  PR[91,1] = PR[90,1] + 48.892;
   1:  PR[91,2] = PR[90,2] + 22.879;
   1:  PR[91,3] = PR[90,3] + 90.750;
   1:L PR[91] R[100]mm/sec CNT100;
   1:  PR[91,1] = PR[90,1] + 47.097;
   1:  PR[91,2] = PR[90,2] + 24.247;
   1:  PR[91,3] = PR[90,3] + 90.763;
   1:L PR[91] R[100]mm/sec CNT100;
   1:  PR[91,1] = PR[90,1] + 42.574;
   1:  PR[91,2] = PR[90,2] + 26.566;
   1:  PR[91,3] = PR[90,3] + 90.773;
   1:L PR[91] R[100]mm/sec CNT100;
   1:  PR[91,1] = PR[90,1] + 37.636;
   1:  PR[91,2] = PR[90,2] + 28.067;
   1:  PR[91,3] = PR[90,3] + 90.795;
   1:L PR[91] R[100]mm/sec CNT100;
   1:  PR[91,1] = PR[90,1] + 32.444;
   1:  PR[91,2] = PR[90,2] + 28.693;
   1:  PR[91,3] = PR[90,3] + 90.817;
   1:L PR[91] R[100]mm/sec CNT100;
   1:  PR[91,1] = PR[90,1] + 27.173;
   1:  PR[91,2] = PR[90,2] + 28.404;
   1:  PR[91,3] = PR[90,3] + 90.840;
   1:L PR[91] R[100]mm/sec CNT100;
   1:  PR[91,1] = PR[90,1] + 21.692;
   1:  PR[91,2] = PR[90,2] + 27.112;
   1:  PR[91,3] = PR[90,3] + 90.863;
   1:L PR[91] R[100]mm/sec CNT100;
   1:  PR[91,1] = PR[90,1] + 19.306;
   1:  PR[91,2] = PR[90,2] + 27.137;
   1:  PR[91,3] = PR[90,3] + 90.888;
   1:L PR[91] R[100]mm/sec CNT100;
   1:  PR[91,1] = PR[90,1] + 18.181;
   1:  PR[91,2] = PR[90,2] + 27.085;
   1:  PR[91,3] = PR[90,3] + 90.898;
   1:L PR[91] R[100]mm/sec CNT100;
   1:  PR[91,1] = PR[90,1] + 16.551;
   1:  PR[91,2] = PR[90,2] + 26.885;
   1:  PR[91,3] = PR[90,3] + 90.903;
   1:L PR[91] R[100]mm/sec CNT100;
   1:  PR[91,1] = PR[90,1] + 15.549;
   1:  PR[91,2] = PR[90,2] + 26.826;
   1:  PR[91,3] = PR[90,3] + 90.910;
   1:L PR[91] R[100]mm/sec CNT100;
   1:  PR[91,1] = PR[90,1] + 13.803;
   1:  PR[91,2] = PR[90,2] + 26.970;
   1:  PR[91,3] = PR[90,3] + 90.914;
   1:L PR[91] R[100]mm/sec CNT100;
   1:  PR[91,1] = PR[90,1] + 12.939;
   1:  PR[91,2] = PR[90,2] + 27.013;
   1:  PR[91,3] = PR[90,3] + 90.922;
   1:L PR[91] R[100]mm/sec CNT100;
   1:  PR[91,1] = PR[90,1] + 8.683;
   1:  PR[91,2] = PR[90,2] + 27.178;
   1:  PR[91,3] = PR[90,3] + 90.926;
   1:L PR[91] R[100]mm/sec CNT100;
   1:  PR[91,1] = PR[90,1] + 2.290;
   1:  PR[91,2] = PR[90,2] + 27.379;
   1:  PR[91,3] = PR[90,3] + 90.944;
   1:L PR[91] R[100]mm/sec CNT100;
   1:  PR[91,1] = PR[90,1] + -8.086;
   1:  PR[91,2] = PR[90,2] + 26.989;
   1:  PR[91,3] = PR[90,3] + 90.972;
   1:L PR[91] R[100]mm/sec CNT100;
   1:  PR[91,1] = PR[90,1] + -12.621;
   1:  PR[91,2] = PR[90,2] + 26.516;
   1:  PR[91,3] = PR[90,3] + 91.018;
   1:L PR[91] R[100]mm/sec CNT100;
   1:  PR[91,1] = PR[90,1] + -17.967;
   1:  PR[91,2] = PR[90,2] + 25.932;
   1:  PR[91,3] = PR[90,3] + 91.037;
   1:L PR[91] R[100]mm/sec CNT100;
   1:  PR[91,1] = PR[90,1] + -27.190;
   1:  PR[91,2] = PR[90,2] + 24.278;
   1:  PR[91,3] = PR[90,3] + 91.061;
   1:L PR[91] R[100]mm/sec CNT100;
   1:  PR[91,1] = PR[90,1] + -35.555;
   1:  PR[91,2] = PR[90,2] + 22.104;
   1:  PR[91,3] = PR[90,3] + 91.102;
   1:L PR[91] R[100]mm/sec CNT100;
   1:  PR[91,1] = PR[90,1] + -40.381;
   1:  PR[91,2] = PR[90,2] + 20.261;
   1:  PR[91,3] = PR[90,3] + 91.139;
   1:L PR[91] R[100]mm/sec CNT100;
   1:  PR[91,1] = PR[90,1] + -45.678;
   1:  PR[91,2] = PR[90,2] + 17.818;
   1:  PR[91,3] = PR[90,3] + 91.162;
   1:L PR[91] R[100]mm/sec CNT100;
   1:  PR[91,1] = PR[90,1] + -46.273;
   1:  PR[91,2] = PR[90,2] + 17.514;
   1:  PR[91,3] = PR[90,3] + 91.187;
   1:L PR[91] R[100]mm/sec CNT100;
   1:  PR[91,1] = PR[90,1] + -47.159;
   1:  PR[91,2] = PR[90,2] + 16.922;
   1:  PR[91,3] = PR[90,3] + 91.190;
   1:L PR[91] R[100]mm/sec CNT100;
   1:  PR[91] = PR[90];
   1:  PR[91,1] = PR[90,1] + -50.121;
   1:  PR[91,2] = PR[90,2] + 13.621;
   1:  PR[91,3] = PR[90,3] + 92.495;
   1:L PR[91] R[100]mm/sec CNT100;
   1:  PR[91,1] = PR[90,1] + -51.090;
   1:  PR[91,2] = PR[90,2] + 12.553;
   1:  PR[91,3] = PR[90,3] + 91.207;
   1:L PR[91] R[100]mm/sec CNT100;
   1:  PR[91,1] = PR[90,1] + -54.051;
   1:  PR[91,2] = PR[90,2] + 9.133;
   1:  PR[91,3] = PR[90,3] + 91.213;
   1:L PR[91] R[100]mm/sec CNT100;
   1:  PR[91,1] = PR[90,1] + -55.580;
   1:  PR[91,2] = PR[90,2] + 6.165;
   1:  PR[91,3] = PR[90,3] + 91.233;
   1:L PR[91] R[100]mm/sec CNT100;
   1:  PR[91,1] = PR[90,1] + -56.502;
   1:  PR[91,2] = PR[90,2] + 4.285;
   1:  PR[91,3] = PR[90,3] + 91.248;
   1:L PR[91] R[100]mm/sec CNT100;
   1:  PR[91,1] = PR[90,1] + -57.148;
   1:  PR[91,2] = PR[90,2] + 0.460;
   1:  PR[91,3] = PR[90,3] + 91.257;
   1:L PR[91] R[100]mm/sec CNT100;
   1:  PR[91,1] = PR[90,1] + -57.399;
   1:  PR[91,2] = PR[90,2] + -0.745;
   1:  PR[91,3] = PR[90,3] + 91.274;
   1:L PR[91] R[100]mm/sec CNT100;
   1:  PR[91,1] = PR[90,1] + -57.058;
   1:  PR[91,2] = PR[90,2] + -2.522;
   1:  PR[91,3] = PR[90,3] + 91.279;
   1:L PR[91] R[100]mm/sec CNT100;
   1:  PR[91,1] = PR[90,1] + -56.883;
   1:  PR[91,2] = PR[90,2] + -2.998;
   1:  PR[91,3] = PR[90,3] + 91.287;
   1:L PR[91] R[100]mm/sec CNT100;
   1:  PR[91,1] = PR[90,1] + -56.485;
   1:  PR[91,2] = PR[90,2] + -5.538;
   1:  PR[91,3] = PR[90,3] + 91.290;
   1:L PR[91] R[100]mm/sec CNT100;
   1:  PR[91,1] = PR[90,1] + -55.562;
   1:  PR[91,2] = PR[90,2] + -7.510;
   1:  PR[91,3] = PR[90,3] + 91.301;
   1:L PR[91] R[100]mm/sec CNT100;
   1:  PR[91,1] = PR[90,1] + -54.199;
   1:  PR[91,2] = PR[90,2] + -10.337;
   1:  PR[91,3] = PR[90,3] + 91.311;
   1:L PR[91] R[100]mm/sec CNT100;
   1:  PR[91,1] = PR[90,1] + -53.264;
   1:  PR[91,2] = PR[90,2] + -11.477;
   1:  PR[91,3] = PR[90,3] + 91.324;
   1:L PR[91] R[100]mm/sec CNT100;
   1:  PR[91,1] = PR[90,1] + -50.242;
   1:  PR[91,2] = PR[90,2] + -15.034;
   1:  PR[91,3] = PR[90,3] + 91.331;
   1:L PR[91] R[100]mm/sec CNT100;
   1:  PR[91,1] = PR[90,1] + -49.453;
   1:  PR[91,2] = PR[90,2] + -15.648;
   1:  PR[91,3] = PR[90,3] + 91.351;
   1:L PR[91] R[100]mm/sec CNT100;
   1:  PR[91,1] = PR[90,1] + -44.605;
   1:  PR[91,2] = PR[90,2] + -18.891;
   1:  PR[91,3] = PR[90,3] + 91.356;
   1:L PR[91] R[100]mm/sec CNT100;
   1:  PR[91,1] = PR[90,1] + -41.813;
   1:  PR[91,2] = PR[90,2] + -20.331;
   1:  PR[91,3] = PR[90,3] + 91.382;
   1:L PR[91] R[100]mm/sec CNT100;
   1:  PR[91,1] = PR[90,1] + -39.127;
   1:  PR[91,2] = PR[90,2] + -21.566;
   1:  PR[91,3] = PR[90,3] + 91.395;
   1:L PR[91] R[100]mm/sec CNT100;
   1:  PR[91,1] = PR[90,1] + -36.152;
   1:  PR[91,2] = PR[90,2] + -22.717;
   1:  PR[91,3] = PR[90,3] + 91.408;
   1:L PR[91] R[100]mm/sec CNT100;
   1:  PR[91,1] = PR[90,1] + -33.238;
   1:  PR[91,2] = PR[90,2] + -23.753;
   1:  PR[91,3] = PR[90,3] + 91.423;
   1:L PR[91] R[100]mm/sec CNT100;
   1:  PR[91,1] = PR[90,1] + -24.786;
   1:  PR[91,2] = PR[90,2] + -25.953;
   1:  PR[91,3] = PR[90,3] + 91.436;
   1:L PR[91] R[100]mm/sec CNT100;
   1:  PR[91,1] = PR[90,1] + -21.549;
   1:  PR[91,2] = PR[90,2] + -26.545;
   1:  PR[91,3] = PR[90,3] + 91.475;
   1:L PR[91] R[100]mm/sec CNT100;
   1:  PR[91,1] = PR[90,1] + -15.498;
   1:  PR[91,2] = PR[90,2] + -27.623;
   1:  PR[91,3] = PR[90,3] + 91.489;
   1:L PR[91] R[100]mm/sec CNT100;
   1:  PR[91,1] = PR[90,1] + -9.208;
   1:  PR[91,2] = PR[90,2] + -28.310;
   1:  PR[91,3] = PR[90,3] + 91.516;
   1:L PR[91] R[100]mm/sec CNT100;
   1:  PR[91,1] = PR[90,1] + -5.540;
   1:  PR[91,2] = PR[90,2] + -28.692;
   1:  PR[91,3] = PR[90,3] + 91.544;
   1:L PR[91] R[100]mm/sec CNT100;
   1:  PR[91,1] = PR[90,1] + 4.915;
   1:  PR[91,2] = PR[90,2] + -29.090;
   1:  PR[91,3] = PR[90,3] + 91.560;
   1:L PR[91] R[100]mm/sec CNT100;
   1:  PR[91,1] = PR[90,1] + 11.842;
   1:  PR[91,2] = PR[90,2] + -28.857;
   1:  PR[91,3] = PR[90,3] + 91.606;
   1:L PR[91] R[100]mm/sec CNT100;
   1:  PR[91,1] = PR[90,1] + 16.065;
   1:  PR[91,2] = PR[90,2] + -28.677;
   1:  PR[91,3] = PR[90,3] + 91.637;
   1:L PR[91] R[100]mm/sec CNT100;
   1:  PR[91,1] = PR[90,1] + 17.327;
   1:  PR[91,2] = PR[90,2] + -28.590;
   1:  PR[91,3] = PR[90,3] + 91.656;
   1:L PR[91] R[100]mm/sec CNT100;
   1:  PR[91,1] = PR[90,1] + 18.267;
   1:  PR[91,2] = PR[90,2] + -28.686;
   1:  PR[91,3] = PR[90,3] + 91.661;
   1:L PR[91] R[100]mm/sec CNT100;
   1:  PR[91,1] = PR[90,1] + 19.931;
   1:  PR[91,2] = PR[90,2] + -28.763;
   1:  PR[91,3] = PR[90,3] + 91.665;
   1:L PR[91] R[100]mm/sec CNT100;
   1:  PR[91,1] = PR[90,1] + 22.994;
   1:  PR[91,2] = PR[90,2] + -28.705;
   1:  PR[91,3] = PR[90,3] + 91.673;
   1:L PR[91] R[100]mm/sec CNT100;
   1:  PR[91,1] = PR[90,1] + 23.074;
   1:  PR[91,2] = PR[90,2] + -29.110;
   1:  PR[91,3] = PR[90,3] + 91.686;
   1:L PR[91] R[100]mm/sec CNT100;
   1:  PR[91,1] = PR[90,1] + 26.769;
   1:  PR[91,2] = PR[90,2] + -29.990;
   1:  PR[91,3] = PR[90,3] + 91.688;
   1:L PR[91] R[100]mm/sec CNT100;
   1:  PR[91,1] = PR[90,1] + 27.259;
   1:  PR[91,2] = PR[90,2] + -30.069;
   1:  PR[91,3] = PR[90,3] + 91.705;
   1:L PR[91] R[100]mm/sec CNT100;
   1:  PR[91,1] = PR[90,1] + 32.225;
   1:  PR[91,2] = PR[90,2] + -30.343;
   1:  PR[91,3] = PR[90,3] + 91.707;
   1:L PR[91] R[100]mm/sec CNT100;
   1:  PR[91,1] = PR[90,1] + 37.453;
   1:  PR[91,2] = PR[90,2] + -29.713;
   1:  PR[91,3] = PR[90,3] + 91.729;
   1:L PR[91] R[100]mm/sec CNT100;
   1:  PR[91,1] = PR[90,1] + 42.429;
   1:  PR[91,2] = PR[90,2] + -28.207;
   1:  PR[91,3] = PR[90,3] + 91.752;
   1:L PR[91] R[100]mm/sec CNT100;
   1:  PR[91,1] = PR[90,1] + 44.848;
   1:  PR[91,2] = PR[90,2] + -26.963;
   1:  PR[91,3] = PR[90,3] + 91.775;
   1:L PR[91] R[100]mm/sec CNT100;
   1:  PR[91,1] = PR[90,1] + 47.005;
   1:  PR[91,2] = PR[90,2] + -25.877;
   1:  PR[91,3] = PR[90,3] + 91.787;
   1:L PR[91] R[100]mm/sec CNT100;
   1:  PR[91,1] = PR[90,1] + 51.024;
   1:  PR[91,2] = PR[90,2] + -22.820;
   1:  PR[91,3] = PR[90,3] + 91.798;
   1:L PR[91] R[100]mm/sec CNT100;
   1:  PR[91,1] = PR[90,1] + 52.149;
   1:  PR[91,2] = PR[90,2] + -21.599;
   1:  PR[91,3] = PR[90,3] + 91.820;
   1:L PR[91] R[100]mm/sec CNT100;
   1:  PR[91,1] = PR[90,1] + 54.553;
   1:  PR[91,2] = PR[90,2] + -19.145;
   1:  PR[91,3] = PR[90,3] + 91.827;
   1:L PR[91] R[100]mm/sec CNT100;
   1:  PR[91,1] = PR[90,1] + 57.366;
   1:  PR[91,2] = PR[90,2] + -15.027;
   1:  PR[91,3] = PR[90,3] + 91.842;
   1:L PR[91] R[100]mm/sec CNT100;
   1:  PR[91,1] = PR[90,1] + 59.402;
   1:  PR[91,2] = PR[90,2] + -10.505;
   1:  PR[91,3] = PR[90,3] + 91.864;
   1:L PR[91] R[100]mm/sec CNT100;
   1:  PR[91,1] = PR[90,1] + 60.496;
   1:  PR[91,2] = PR[90,2] + -6.223;
   1:  PR[91,3] = PR[90,3] + 91.886;
   1:L PR[91] R[100]mm/sec CNT100;
   1:  PR[91,1] = PR[90,1] + 60.661;
   1:  PR[91,2] = PR[90,2] + -5.644;
   1:  PR[91,3] = PR[90,3] + 91.906;
   1:L PR[91] R[100]mm/sec CNT100;
   1:  PR[91,1] = PR[90,1] + 61.112;
   1:  PR[91,2] = PR[90,2] + -0.706;
   1:  PR[91,3] = PR[90,3] + 91.908;
   1:L PR[91] R[100]mm/sec CNT100;
   1:  PR[91,1] = PR[90,1] + 61.095;
   1:  PR[91,2] = PR[90,2] + -0.444;
   1:  PR[91,3] = PR[90,3] + 91.930;
   1:L PR[91] R[100]mm/sec CNT100;
   1:  PR[91,1] = PR[90,1] + 60.662;
   1:  PR[91,2] = PR[90,2] + 4.183;
   1:  PR[91,3] = PR[90,3] + 91.931;
   1:L PR[91] R[100]mm/sec CNT100;
   1:  PR[91,1] = PR[90,1] + 60.496;
   1:  PR[91,2] = PR[90,2] + 4.764;
   1:  PR[91,3] = PR[90,3] + 91.952;
   1:L PR[91] R[100]mm/sec CNT100;
   1:  PR[91,1] = PR[90,1] + 59.402;
   1:  PR[91,2] = PR[90,2] + 9.046;
   1:  PR[91,3] = PR[90,3] + 91.954;
   1:L PR[91] R[100]mm/sec CNT100;
   1:  PR[91,1] = PR[90,1] + 57.365;
   1:  PR[91,2] = PR[90,2] + 13.568;
   1:  PR[91,3] = PR[90,3] + 91.974;
   1:L PR[91] R[100]mm/sec CNT100;
   1:  PR[91,1] = PR[90,1] + 54.553;
   1:  PR[91,2] = PR[90,2] + 17.686;
   1:  PR[91,3] = PR[90,3] + 91.996;
   1:L PR[91] R[100]mm/sec CNT100;
   1:  PR[91,1] = PR[90,1] + 52.149;
   1:  PR[91,2] = PR[90,2] + 20.140;
   1:  PR[91,3] = PR[90,3] + 92.018;
   1:L PR[91] R[100]mm/sec CNT100;
   1:  PR[91,1] = PR[90,1] + 51.024;
   1:  PR[91,2] = PR[90,2] + 21.361;
   1:  PR[91,3] = PR[90,3] + 92.033;
   1:L PR[91] R[100]mm/sec CNT100;
   1:  PR[91,1] = PR[90,1] + 47.005;
   1:  PR[91,2] = PR[90,2] + 24.418;
   1:  PR[91,3] = PR[90,3] + 92.040;
   1:L PR[91] R[100]mm/sec CNT100;
   1:  PR[91,1] = PR[90,1] + 44.848;
   1:  PR[91,2] = PR[90,2] + 25.504;
   1:  PR[91,3] = PR[90,3] + 92.062;
   1:L PR[91] R[100]mm/sec CNT100;
   1:  PR[91,1] = PR[90,1] + 42.429;
   1:  PR[91,2] = PR[90,2] + 26.748;
   1:  PR[91,3] = PR[90,3] + 92.073;
   1:L PR[91] R[100]mm/sec CNT100;
   1:  PR[91,1] = PR[90,1] + 37.453;
   1:  PR[91,2] = PR[90,2] + 28.254;
   1:  PR[91,3] = PR[90,3] + 92.085;
   1:L PR[91] R[100]mm/sec CNT100;
   1:  PR[91,1] = PR[90,1] + 32.225;
   1:  PR[91,2] = PR[90,2] + 28.884;
   1:  PR[91,3] = PR[90,3] + 92.108;
   1:L PR[91] R[100]mm/sec CNT100;
   1:  PR[91,1] = PR[90,1] + 27.261;
   1:  PR[91,2] = PR[90,2] + 28.611;
   1:  PR[91,3] = PR[90,3] + 92.131;
   1:L PR[91] R[100]mm/sec CNT100;
   1:  PR[91,1] = PR[90,1] + 26.766;
   1:  PR[91,2] = PR[90,2] + 28.530;
   1:  PR[91,3] = PR[90,3] + 92.153;
   1:L PR[91] R[100]mm/sec CNT100;
   1:  PR[91,1] = PR[90,1] + 21.551;
   1:  PR[91,2] = PR[90,2] + 27.288;
   1:  PR[91,3] = PR[90,3] + 92.155;
   1:L PR[91] R[100]mm/sec CNT100;
   1:  PR[91,1] = PR[90,1] + 19.940;
   1:  PR[91,2] = PR[90,2] + 27.304;
   1:  PR[91,3] = PR[90,3] + 92.179;
   1:L PR[91] R[100]mm/sec CNT100;
   1:  PR[91,1] = PR[90,1] + 18.289;
   1:  PR[91,2] = PR[90,2] + 27.228;
   1:  PR[91,3] = PR[90,3] + 92.186;
   1:L PR[91] R[100]mm/sec CNT100;
   1:  PR[91,1] = PR[90,1] + 17.745;
   1:  PR[91,2] = PR[90,2] + 27.162;
   1:  PR[91,3] = PR[90,3] + 92.193;
   1:L PR[91] R[100]mm/sec CNT100;
   1:  PR[91,1] = PR[90,1] + 17.271;
   1:  PR[91,2] = PR[90,2] + 27.133;
   1:  PR[91,3] = PR[90,3] + 92.196;
   1:L PR[91] R[100]mm/sec CNT100;
   1:  PR[91,1] = PR[90,1] + 16.605;
   1:  PR[91,2] = PR[90,2] + 27.189;
   1:  PR[91,3] = PR[90,3] + 92.198;
   1:L PR[91] R[100]mm/sec CNT100;
   1:  PR[91,1] = PR[90,1] + 15.610;
   1:  PR[91,2] = PR[90,2] + 27.240;
   1:  PR[91,3] = PR[90,3] + 92.201;
   1:L PR[91] R[100]mm/sec CNT100;
   1:  PR[91,1] = PR[90,1] + 8.035;
   1:  PR[91,2] = PR[90,2] + 27.533;
   1:  PR[91,3] = PR[90,3] + 92.205;
   1:L PR[91] R[100]mm/sec CNT100;
   1:  PR[91,1] = PR[90,1] + 4.917;
   1:  PR[91,2] = PR[90,2] + 27.632;
   1:  PR[91,3] = PR[90,3] + 92.239;
   1:L PR[91] R[100]mm/sec CNT100;
   1:  PR[91,1] = PR[90,1] + -5.540;
   1:  PR[91,2] = PR[90,2] + 27.233;
   1:  PR[91,3] = PR[90,3] + 92.252;
   1:L PR[91] R[100]mm/sec CNT100;
   1:  PR[91,1] = PR[90,1] + -9.208;
   1:  PR[91,2] = PR[90,2] + 26.851;
   1:  PR[91,3] = PR[90,3] + 92.298;
   1:L PR[91] R[100]mm/sec CNT100;
   1:  PR[91,1] = PR[90,1] + -15.498;
   1:  PR[91,2] = PR[90,2] + 26.164;
   1:  PR[91,3] = PR[90,3] + 92.315;
   1:L PR[91] R[100]mm/sec CNT100;
   1:  PR[91,1] = PR[90,1] + -21.549;
   1:  PR[91,2] = PR[90,2] + 25.086;
   1:  PR[91,3] = PR[90,3] + 92.343;
   1:L PR[91] R[100]mm/sec CNT100;
   1:  PR[91,1] = PR[90,1] + -24.786;
   1:  PR[91,2] = PR[90,2] + 24.494;
   1:  PR[91,3] = PR[90,3] + 92.370;
   1:L PR[91] R[100]mm/sec CNT100;
   1:  PR[91,1] = PR[90,1] + -33.238;
   1:  PR[91,2] = PR[90,2] + 22.294;
   1:  PR[91,3] = PR[90,3] + 92.384;
   1:L PR[91] R[100]mm/sec CNT100;
   1:  PR[91,1] = PR[90,1] + -36.156;
   1:  PR[91,2] = PR[90,2] + 21.257;
   1:  PR[91,3] = PR[90,3] + 92.423;
   1:L PR[91] R[100]mm/sec CNT100;
   1:  PR[91,1] = PR[90,1] + -39.108;
   1:  PR[91,2] = PR[90,2] + 20.129;
   1:  PR[91,3] = PR[90,3] + 92.436;
   1:L PR[91] R[100]mm/sec CNT100;
   1:  PR[91,1] = PR[90,1] + -42.315;
   1:  PR[91,2] = PR[90,2] + 18.650;
   1:  PR[91,3] = PR[90,3] + 92.450;
   1:L PR[91] R[100]mm/sec CNT100;
   1:  PR[91,1] = PR[90,1] + -44.657;
   1:  PR[91,2] = PR[90,2] + 17.456;
   1:  PR[91,3] = PR[90,3] + 92.466;
   1:L PR[91] R[100]mm/sec CNT100;
   1:  PR[91,1] = PR[90,1] + -47.997;
   1:  PR[91,2] = PR[90,2] + 15.223;
   1:  PR[91,3] = PR[90,3] + 92.477;
   1:L PR[91] R[100]mm/sec CNT100;
   1:  PR[91] = PR[90];
   1:  PR[91,1] = PR[90,1] + -52.602;
   1:  PR[91,2] = PR[90,2] + 9.120;
   1:  PR[91,3] = PR[90,3] + 93.795;
   1:L PR[91] R[100]mm/sec CNT100;
   1:  PR[91,1] = PR[90,1] + -53.557;
   1:  PR[91,2] = PR[90,2] + 7.266;
   1:  PR[91,3] = PR[90,3] + 92.521;
   1:L PR[91] R[100]mm/sec CNT100;
   1:  PR[91,1] = PR[90,1] + -55.024;
   1:  PR[91,2] = PR[90,2] + 4.276;
   1:  PR[91,3] = PR[90,3] + 92.531;
   1:L PR[91] R[100]mm/sec CNT100;
   1:  PR[91,1] = PR[90,1] + -55.498;
   1:  PR[91,2] = PR[90,2] + 1.469;
   1:  PR[91,3] = PR[90,3] + 92.545;
   1:L PR[91] R[100]mm/sec CNT100;
   1:  PR[91,1] = PR[90,1] + -55.960;
   1:  PR[91,2] = PR[90,2] + -0.745;
   1:  PR[91,3] = PR[90,3] + 92.558;
   1:L PR[91] R[100]mm/sec CNT100;
   1:  PR[91,1] = PR[90,1] + -55.785;
   1:  PR[91,2] = PR[90,2] + -1.653;
   1:  PR[91,3] = PR[90,3] + 92.568;
   1:L PR[91] R[100]mm/sec CNT100;
   1:  PR[91,1] = PR[90,1] + -55.561;
   1:  PR[91,2] = PR[90,2] + -2.263;
   1:  PR[91,3] = PR[90,3] + 92.572;
   1:L PR[91] R[100]mm/sec CNT100;
   1:  PR[91,1] = PR[90,1] + -55.038;
   1:  PR[91,2] = PR[90,2] + -5.599;
   1:  PR[91,3] = PR[90,3] + 92.575;
   1:L PR[91] R[100]mm/sec CNT100;
   1:  PR[91,1] = PR[90,1] + -54.426;
   1:  PR[91,2] = PR[90,2] + -6.908;
   1:  PR[91,3] = PR[90,3] + 92.590;
   1:L PR[91] R[100]mm/sec CNT100;
   1:  PR[91,1] = PR[90,1] + -52.715;
   1:  PR[91,2] = PR[90,2] + -10.457;
   1:  PR[91,3] = PR[90,3] + 92.597;
   1:L PR[91] R[100]mm/sec CNT100;
   1:  PR[91,1] = PR[90,1] + -52.268;
   1:  PR[91,2] = PR[90,2] + -11.002;
   1:  PR[91,3] = PR[90,3] + 92.614;
   1:L PR[91] R[100]mm/sec CNT100;
   1:  PR[91,1] = PR[90,1] + -50.009;
   1:  PR[91,2] = PR[90,2] + -13.661;
   1:  PR[91,3] = PR[90,3] + 92.617;
   1:L PR[91] R[100]mm/sec CNT100;
   1:  PR[91,1] = PR[90,1] + -48.814;
   1:  PR[91,2] = PR[90,2] + -14.872;
   1:  PR[91,3] = PR[90,3] + 92.633;
   1:L PR[91] R[100]mm/sec CNT100;
   1:  PR[91,1] = PR[90,1] + -48.612;
   1:  PR[91,2] = PR[90,2] + -15.066;
   1:  PR[91,3] = PR[90,3] + 92.640;
   1:L PR[91] R[100]mm/sec CNT100;
   1:  PR[91,1] = PR[90,1] + -47.915;
   1:  PR[91,2] = PR[90,2] + -15.552;
   1:  PR[91,3] = PR[90,3] + 92.642;
   1:L PR[91] R[100]mm/sec CNT100;
   1:  PR[91,1] = PR[90,1] + -43.001;
   1:  PR[91,2] = PR[90,2] + -18.839;
   1:  PR[91,3] = PR[90,3] + 92.645;
   1:L PR[91] R[100]mm/sec CNT100;
   1:  PR[91,1] = PR[90,1] + -38.766;
   1:  PR[91,2] = PR[90,2] + -21.024;
   1:  PR[91,3] = PR[90,3] + 92.672;
   1:L PR[91] R[100]mm/sec CNT100;
   1:  PR[91,1] = PR[90,1] + -37.840;
   1:  PR[91,2] = PR[90,2] + -21.449;
   1:  PR[91,3] = PR[90,3] + 92.693;
   1:L PR[91] R[100]mm/sec CNT100;
   1:  PR[91,1] = PR[90,1] + -36.800;
   1:  PR[91,2] = PR[90,2] + -21.851;
   1:  PR[91,3] = PR[90,3] + 92.698;
   1:L PR[91] R[100]mm/sec CNT100;
   1:  PR[91,1] = PR[90,1] + -30.899;
   1:  PR[91,2] = PR[90,2] + -23.948;
   1:  PR[91,3] = PR[90,3] + 92.702;
   1:L PR[91] R[100]mm/sec CNT100;
   1:  PR[91,1] = PR[90,1] + -22.384;
   1:  PR[91,2] = PR[90,2] + -26.169;
   1:  PR[91,3] = PR[90,3] + 92.730;
   1:L PR[91] R[100]mm/sec CNT100;
   1:  PR[91,1] = PR[90,1] + -18.279;
   1:  PR[91,2] = PR[90,2] + -26.920;
   1:  PR[91,3] = PR[90,3] + 92.770;
   1:L PR[91] R[100]mm/sec CNT100;
   1:  PR[91,1] = PR[90,1] + -13.027;
   1:  PR[91,2] = PR[90,2] + -27.855;
   1:  PR[91,3] = PR[90,3] + 92.788;
   1:L PR[91] R[100]mm/sec CNT100;
   1:  PR[91,1] = PR[90,1] + -5.796;
   1:  PR[91,2] = PR[90,2] + -28.645;
   1:  PR[91,3] = PR[90,3] + 92.812;
   1:L PR[91] R[100]mm/sec CNT100;
   1:  PR[91,1] = PR[90,1] + -2.993;
   1:  PR[91,2] = PR[90,2] + -28.937;
   1:  PR[91,3] = PR[90,3] + 92.844;
   1:L PR[91] R[100]mm/sec CNT100;
   1:  PR[91,1] = PR[90,1] + 7.528;
   1:  PR[91,2] = PR[90,2] + -29.343;
   1:  PR[91,3] = PR[90,3] + 92.857;
   1:L PR[91] R[100]mm/sec CNT100;
   1:  PR[91,1] = PR[90,1] + 12.860;
   1:  PR[91,2] = PR[90,2] + -29.154;
   1:  PR[91,3] = PR[90,3] + 92.904;
   1:L PR[91] R[100]mm/sec CNT100;
   1:  PR[91,1] = PR[90,1] + 18.504;
   1:  PR[91,2] = PR[90,2] + -28.915;
   1:  PR[91,3] = PR[90,3] + 92.927;
   1:L PR[91] R[100]mm/sec CNT100;
   1:  PR[91,1] = PR[90,1] + 19.231;
   1:  PR[91,2] = PR[90,2] + -28.869;
   1:  PR[91,3] = PR[90,3] + 92.952;
   1:L PR[91] R[100]mm/sec CNT100;
   1:  PR[91,1] = PR[90,1] + 20.565;
   1:  PR[91,2] = PR[90,2] + -28.931;
   1:  PR[91,3] = PR[90,3] + 92.956;
   1:L PR[91] R[100]mm/sec CNT100;
   1:  PR[91,1] = PR[90,1] + 22.832;
   1:  PR[91,2] = PR[90,2] + -28.888;
   1:  PR[91,3] = PR[90,3] + 92.962;
   1:L PR[91] R[100]mm/sec CNT100;
   1:  PR[91,1] = PR[90,1] + 22.910;
   1:  PR[91,2] = PR[90,2] + -29.281;
   1:  PR[91,3] = PR[90,3] + 92.972;
   1:L PR[91] R[100]mm/sec CNT100;
   1:  PR[91,1] = PR[90,1] + 26.167;
   1:  PR[91,2] = PR[90,2] + -30.059;
   1:  PR[91,3] = PR[90,3] + 92.974;
   1:L PR[91] R[100]mm/sec CNT100;
   1:  PR[91,1] = PR[90,1] + 27.564;
   1:  PR[91,2] = PR[90,2] + -30.285;
   1:  PR[91,3] = PR[90,3] + 92.988;
   1:L PR[91] R[100]mm/sec CNT100;
   1:  PR[91,1] = PR[90,1] + 31.764;
   1:  PR[91,2] = PR[90,2] + -30.517;
   1:  PR[91,3] = PR[90,3] + 92.995;
   1:L PR[91] R[100]mm/sec CNT100;
   1:  PR[91,1] = PR[90,1] + 32.510;
   1:  PR[91,2] = PR[90,2] + -30.502;
   1:  PR[91,3] = PR[90,3] + 93.013;
   1:L PR[91] R[100]mm/sec CNT100;
   1:  PR[91,1] = PR[90,1] + 37.245;
   1:  PR[91,2] = PR[90,2] + -29.906;
   1:  PR[91,3] = PR[90,3] + 93.017;
   1:L PR[91] R[100]mm/sec CNT100;
   1:  PR[91,1] = PR[90,1] + 42.292;
